hm	1. okt 2007		rev 1.1
	added compatibility to STEP7

*)
END_FUNCTION

(* POU leap_of_Date, ST *)
FUNCTION leap_of_Date : BOOL
VAR_INPUT
	idate : DATE;
END_VAR
VAR
END_VAR

(*
version 1.1	2 oct 2006
programmer 	hugo
tested by		tobias


leap_year is true if the tested year is a leap year  
execution time on wago 750-841 =  30 us   
*)
leap_of_Date := leap_year(year(idate));


(* change history

2.10.2006		changes to rev 1.1
the function now calls leap_year to accomodate further accuracy.
the function now works for any year from 1970 to 2100

*)
END_FUNCTION

(* POU leap_year, ST *)
FUNCTION leap_year : BOOL
VAR_INPUT
	yr : INT;
END_VAR
VAR
END_VAR

(*
version 1.1	2 oct 2006
programmer 	hugo
tested by		tobias


leap_year is true if the tested year is a leap year  
execution time on wago 750-841 =  12 us    
*)
leap_year := SHL(yr,14) = 0;

(* this code was used prior to rev 1.1

IF yr MOD 400 = 0 THEN leap_year := TRUE;
ELSIF yr MOD 100 = 0 THEN leap_year := FALSE;
ELSIF yr MOD 4 =0 THEN leap_year := TRUE;
ELSE leap_year := FALSE;
END_IF;

*)

(* change history

hm 	2.10.2006		rev 1.1
	the function now works for any year from 1970 up to 2100

hm	1. oct 2007		rev 1.2
	chaged code for higher performance
*)
END_FUNCTION

(* POU set_Date, ST *)
FUNCTION set_Date : DATE
VAR_INPUT
	year : INT;
	month : INT;
	day : INT;
END_VAR
VAR
	count : DWORD;
	leap: BOOL;
END_VAR

(*
version 1.2	1 okt 2007
programmer 	hugo
tested by		tobias

creates a date output from year, month and day of month   

*)
leap := leap_year(year);
IF STEP7 THEN
	count := TRUNC((year-1)*365.25-726483+day);
ELSE
	count := TRUNC((year-1)*365.25-719178+day);
END_IF;
CASE month OF
2:	count := count + 31;
3:	IF leap THEN count := count + 60; ELSE count := count + 59; END_IF;
4:	IF leap THEN count := count + 91; ELSE count := count + 90; END_IF;
5:	IF leap THEN count := count + 121; ELSE count := count + 120; END_IF;
6:	IF leap THEN count := count + 152; ELSE count := count + 151; END_IF;
7:	IF leap THEN count := count + 182; ELSE count := count + 181; END_IF;
8:	IF leap THEN count := count + 213; ELSE count := count + 212; END_IF;
9:	IF leap THEN count := count + 244; ELSE count := count + 243; END_IF;
10:	IF leap THEN count := count + 274; ELSE count := count + 273; END_IF;
11:	IF leap THEN count := count + 305; ELSE count := count + 304; END_IF;
12:	IF leap THEN count := count + 335; ELSE count := count + 334; END_IF;
END_CASE;
set_Date := DWORD_TO_DATE(count * 86400);


(* revision history
hm	4. aug. 2006	rev 1.0
	original version

hm	19 sep. 2007	rev 1.1
	use function leap_year to calculate leap year, more exceptions are handled

hm	1. okt	2007	rev 1.2
	added compatibilkity to step7
*)
END_FUNCTION

(* POU day_of_month, ST *)
FUNCTION day_of_month : INT
VAR_INPUT
	idate : DATE;
END_VAR
VAR
	yd: INT;
END_VAR

(*
version 1.3	8. okt 2007
programmer 	hugo
tested by		tobias

returns the day OF month for any DATE

*)
yd := day_of_year(idate);
IF leap_of_Date(idate) THEN
	CASE yd OF
		1..31 	:	day_of_month := yd;
		32..60	:	day_of_month := yd - 31;
		61..91	:	day_of_month := yd - 60;
		92..121 :	day_of_month := yd - 91;
		122..152:	day_of_month := yd - 121;
		153..182:	day_of_month := yd - 152;
		183..213:	day_of_month := yd - 182;
		214..244:	day_of_month := yd - 213;
		245..274:	day_of_month := yd - 244;
		275..305:	day_of_month := yd - 274;
		306..335:	day_of_month := yd - 305;
		336..366:	day_of_month := yd - 335;
	END_CASE;
ELSE
	CASE yd OF
		1..31 	:	day_of_month := yd;
		32..59	:	day_of_month := yd - 31;
		60..90	:	day_of_month := yd - 59;
		91..120 :	day_of_month := yd - 90;
		121..151:	day_of_month := yd - 120;
		152..181:	day_of_month := yd - 151;
		182..212:	day_of_month := yd - 181;
		213..243:	day_of_month := yd - 212;
		244..273:	day_of_month := yd - 243;
		274..304:	day_of_month := yd - 273;
		305..334:	day_of_month := yd - 304;
		335..365:	day_of_month := yd - 334;
	END_CASE;
END_IF;


(*
this function is simple but took too long with 133 us
the problem is date_to_string is far too slow
day_of_month := STRING_TO_INT(RIGHT(DATE_TO_STRING(idate),2));

Revision history

hm 22.1.2007		rev 1.1
	deleted unused variable day_in_year and day_in_year_begin

hm	1. okt 2007		rev 1.2
	changed code to use day_of_year and leap_of_date
	added compatibility to STEP7

hm	8. oct 2007		rev 1.3
	deleted unused variable yr
*)
END_FUNCTION

(* POU days_delta, ST *)
FUNCTION days_delta : INT
VAR_INPUT
	date_1 : DATE;
	date_2 : DATE;
END_VAR
VAR
END_VAR

(*
version 1.1	27 dec 2006
programmer 	hugo
tested by		tobias

days_delta calculates the days between two dates. the days are calculated date_2 - date_1.

*)
days_delta := day_of_date(date_2) - day_of_date(date_1);

(* revision history
hm	27. dec 2006	rev 1.0
	original version

hm	16.9.2007		rev 1.1
	coorected an error in formula and changed algorithm to show positive and negative delta

*)
END_FUNCTION

(* POU day_of_date, ST *)
FUNCTION day_of_date : INT
VAR_INPUT
	idate : DATE;
END_VAR
VAR
END_VAR


(*
	version 1.0	16 sep 2007
	programmer 	oscat
	tested BY		oscat

DAY_OF_DATE returns the days since 1.1.1970

*)
IF STEP7 THEN
	(* adjust step7 day by 7305 days because step7 date fornat starts at 1.1.1990  *)
	day_of_date := DWORD_TO_INT(DATE_TO_DWORD(idate) / 86400) + 7305;
ELSE
	day_of_date := DWORD_TO_INT(DATE_TO_DWORD(idate) / 86400);
END_IF;
(* revision history
hm		16.9.2007		rev 1.0
	original version

hm		1. okt 2007		rev 1.1
	added step7 compatibility

*)
END_FUNCTION

(* POU DST, ST *)
FUNCTION DST : BOOL
VAR_INPUT
	utc : DT;
	time_zone_offset : TIME;
END_VAR
VAR
	yr : INT;
	yr4 : DWORD;
	ltc: DWORD;
	idate : DWORD;
END_VAR

(*
version 1.0	4 aug 2006
programmer 	hugo
tested by		tobias

 this functions returns TRUE IF dst TIME is active 
 the FUNCTION calculates automaticall FOR any year betweek 1970 AND 2099 
wheather daylight savings is on OR off 
the summertime calculation is done according to european standards.
dst will become TRUE AT 02:00 in the morning FOR the respective days 
AND it will become FALSE after daylight savings TIME is switched back end OF october automatically 
(execution TIME on wago 750-841 =  110us   
*)
yr := year(DT_TO_DATE(utc));
ltc := DT_TO_DWORD(utc+time_zone_offset);
idate := DT_TO_DWORD(set_DT(yr,3,31,2,0,0));
yr4 := 5*yr/4;
IF idate - ((yr4+4) MOD 7)*86400 <= ltc AND idate + (214 - (yr4+1) MOD 7)*86400 > ltc THEN DST := TRUE; ELSE DST := FALSE; END_IF;


(*

Equation used TO calculate the beginning OF European Summer TIME:
Sunday (31 - (5*y/4 + 4) mod 7) March at 01.00 UTC
(valid through 2099, courtesy of Robert H. van Gent, EC).

European Summer Time ends (clocks go back) at 01.00 UTC on

    * 29 October 2006
    * 28 October 2007
    * 26 October 2008

Equation used to calculate the end of European Summer Time:
Sunday (31 - (5*y/4 + 1) mod 7) October at 01.00 UTC
(validity AND credits as above).

*)
END_FUNCTION

(* POU set_DT, ST *)
FUNCTION set_DT : DT
VAR_INPUT
	year : INT;
	month : INT;
	day : INT;
	hour : INT;
	minute : INT;
	second : INT;
END_VAR
VAR
END_VAR

(*
version 1.3	8 okt 2007
programmer 	hugo
tested by		tobias


creates a date output from year, month and day of month
year must be in the form of 4 digits ie 2006 or 1977.
execution time on wago 750-841 = 45 us   
*)
set_DT := DWORD_TO_DT(DATE_TO_DWORD(set_Date(year, month, day)) + second + minute * 60 + hour * 3600);


(* revision history
hm	4. aug. 2006	rev 1.0
	original version

hm	19 sep. 2007	rev 1.1
	use function leap_year to calculate leap year, more exceptions are handled

hm	1. okt 2007		rev 1.2
	added step7 compatibility
	call function set_date

hm	8. oct 2007		rev 1.3
	deleted unused variables count and leap
*)
END_FUNCTION

(* POU hour, ST *)
FUNCTION hour : INT
VAR_INPUT
	itod : TOD;
END_VAR
VAR
END_VAR

(*
version 1.1	2 okt 2006
programmer 	hugo
tested by		tobias

extracts the hour of a Time_of_day 
*)
hour := DWORD_TO_INT(TOD_TO_DWORD(itod)/3600000);


(* change history
hm 4. aug 2006	rev 1.0
	original version

hm 2.10.2006 	rev 1.1
	changed name of input to itod

*)
END_FUNCTION

(* POU minute, ST *)
FUNCTION minute : INT
VAR_INPUT
	itod : TOD;
END_VAR
VAR
END_VAR

(*
version 1.1	2 oct 2006
programmer 	hugo
tested by		tobias

extracts the minutes out of TOD truncating the ceconds 
execution time on wago 750-841  = 18us

*)  
minute := DWORD_TO_INT(TOD_TO_DWORD(itod)/60000 - TOD_TO_DWORD(itod)/3600000 * 60);


(* change history

2.10.2006 changes name of input to itod

*)
END_FUNCTION

(* POU second, ST *)
FUNCTION second : REAL
VAR_INPUT
	itod : TOD;
END_VAR
VAR
END_VAR

(*
version 1.1	2 oct 2006
programmer 	hugo
tested by		tobias

returns the seconds and milliseconds as real of TOD   
execution time on wago 750-841 = 20 us 
*)
second := DWORD_TO_REAL(TOD_TO_DWORD(itod) - TOD_TO_DWORD(itod)/60000 * 60000)/1000;



(* change history

2.10.2006 changes name of input to itod

*)
END_FUNCTION

(* POU easter, ST *)
FUNCTION easter : DATE
VAR_INPUT
	year : INT;
END_VAR
VAR
	A: INT;
	B: INT;
	C: INT;
	D: INT;
	e: INT;
	f: INT;
	g: INT;
	h: INT;
	i: INT;
	k: INT;
	l: INT;
	m: INT;
	n: INT;
	o: INT;
END_VAR

(*
version 1.0	27 dec 2006
programmer 	hugo
tested by		tobias

easter calculates the day of easter sunday for a given year.
most other catholic holidays are calculated in reference to easter sunday.

*)
a := year MOD 19;
b := year / 100;
c := year MOD 100;
d := b / 4;
e := b MOD 4;
f :=	(b + 8) / 25;
g := (b - f + 1) / 3;
h := (19 * a + b - d - g + 15) MOD 30;
i :=	c / 4;
k := c MOD 4;
l := (32 + 2 * e + 2 * i - h - k) MOD 7;
m := (a + 11 * h + 22 * l) / 451;
n := (h + l - 7 * m + 114) / 31;
o := (h + l - 7 * m + 114) MOD 31;

easter := set_Date(year,n,o+1);

(*
Im Magazin "Nature" vom 20. April 1876 veröffentlichte ein anonymer Autor eine Tabelle mit Regeln zur Berechnung des (Gregorianischen) Ostersonntages des Jahres J. In Formeln ausgedrückt erhält man das Folgende:
a	=	J mod 19
b	=	int(J / 100)
c	=	J mod 100
d	=	int(b / 4)
e	=	b mod 4
f	=	int((b + 8) / 25)
g	=	int((b - f + 1) / 3
h	=	(19 · a + b - d - g + 15) mod 30
i	=	int(c / 4)
k	=	c mod 4
l	=	(32 + 2 · e + 2 · i - h - k) mod 7
m	=	int((a + 11 · h + 22 · l) / 451)
n	=	int((h + l - 7 · m + 114) / 31)
o	=	(h + l - 7 · m + 114) mod 31

n ist hierbei die Nummer des Monats, o + 1 die Nummer des Tages auf welchen der Ostersonntag im Jahr J fällt. Dieser Algorithmus kommt ohne Hilfszahlen aus.

*)
END_FUNCTION

(* POU hour_to_time, ST *)
FUNCTION hour_to_time : TIME
VAR_INPUT
	input : REAL;
END_VAR
VAR
END_VAR

(*
version 1.0	4 aug 2006
programmer 	hugo
tested by		tobias

converts an amount of hours in real to time
execution TIME on wago 750-841 =  17us
*)
hour_to_time := DWORD_TO_TIME(REAL_TO_DWORD(input * 3600000));
END_FUNCTION

(* POU hour_to_tod, ST *)
FUNCTION hour_to_tod : TOD
VAR_INPUT
	input : REAL;
END_VAR
VAR
END_VAR

(*
version 1.0	4 aug 2006
programmer 	hugo
tested by		tobias

converts an amount of hours in real to time of day 
execution time on wago 750-841 =  17us 
*)
hour_to_tod := DWORD_TO_TOD(REAL_TO_DWORD(input * 3600000));
END_FUNCTION

(* POU local_time, ST *)
FUNCTION local_time : DT
VAR_INPUT
	utc : DT;
	time_zone_offset : TIME;
	dst_enable: BOOL;
END_VAR
VAR
END_VAR

(*
version 1.1	2 oct 2006
programmer 	hugo
tested by		tobias

localtime calculates the local time according to DSTenable and time_zone_offset.
the dst input only tells the function the dst (daylight savings time) is enabled but the calculation for summertime on and off is done by the function itself.
this means the dst input only tells the function to switch summertime on and off automatically or not.
the function will switch to summertime automatically at the specified time end of march and back end of october.
the summertime calculation is done according to european standards.
the input is world time (UTC) and a given time_zone_offset for any time_zone.

execution time on wago 750-841 = 140 us   
*)
IF DST(utc,time_zone_offset) AND dst_enable THEN
	local_time := utc + time_zone_offset + T#1h;
ELSE
	local_time := utc + time_zone_offset;
END_IF;


(*

change history

2.10.2006 hm	rev 1.1
	corrected an error in the dst check for correct function

*)
END_FUNCTION

(* POU Ltime_to_UTC, ST *)
FUNCTION Ltime_to_UTC : DT
VAR_INPUT
	Ltime : DT;
	DST : BOOL;
	Time_Zone_Offset : TIME;
END_VAR
VAR
END_VAR

(*
version 1.0	5 jul 2007
programmer 	hugo
tested by		tobias

LTIME_TO_UTC calculates UTC (World Time) from a local time LTIME. utc is calculated by subtracting Time_Zone_Offset from ltime and if dst it true subtracting an additional hour from ltime.

*)
IF DST THEN Ltime_to_UTC := Ltime - Time_Zone_Offset - t#1h; ELSE Ltime_to_UTC := Ltime - Time_Zone_Offset; END_IF;



(* revision history
5.7.2007	rev 1.0		original version

*)
END_FUNCTION

(* POU Ltime, ST *)
FUNCTION_BLOCK Ltime
VAR_INPUT
	UTC : DT;
	dst_enable : BOOL;
	time_zone_offset : TIME;
END_VAR
VAR_OUTPUT
	local_DT : DT;
	DST_on : BOOL;
	wday : INT;
END_VAR
VAR
	time_adder : TIME := t#0s;
	next_check : DT := dt#1970-01-01-00:00:00;
	init: BOOL;
END_VAR

(*

version 1.3	18 Mar 2007
programmer 	oscat
tested by		tobias

ltime is a real time clock that uses the system rtc as utc time and calculates and given time zone.
the utc time is supplied on the input UTC.
according to the input variable time_zone_offset when the input dst_enable is true,
the dst on and off times are calculated by a formula for any given year and the time is advanced and reset by one hour
at 02:00 and 03:00 for the last sunday of march and last sunday of october.
the code is high performance and the rtc counts every second.
if more then one time zone is needed by the systen the clock can be started many times by placing more then one function block.

execution time on wago 750-841 = 20 us 
 
*)
IF utc > next_check THEN
	IF NOT init THEN
		local_dt := utc + time_zone_offset;
		init := TRUE;
	END_IF;
	next_check := DWORD_TO_DT(DT_TO_DWORD(utc) / 3600 * 3600 +3600);
	DST_on := DST(local_dt, time_zone_offset);
	IF DST_on AND dst_enable THEN time_adder := time_zone_offset + T#1h; ELSE time_adder := time_zone_offset; END_IF;
END_IF;
local_dt :=utc + time_adder;
wday := weekday(DT_TO_DATE(local_dt));

(* revision history

hm 2.10.2006	rev 1.1
	corrected an error where dst would be delayed by 0.1second

hm 17.1.2007	rev 1.2
	added utc input instead of internal sysrtcgettime because this would only work on wago.
	dst_enable would not be checked before dst would be enabled.

hm 18.3.2007	rev 1.3
	changed code, dst would not work during first cycle.

*)
END_FUNCTION_BLOCK

(* POU weekday, ST *)
FUNCTION weekday : INT
VAR_INPUT
	idate : DATE;
END_VAR
VAR
END_VAR

(*
version 1.1	21 aug 2006
programmer 	hugo
tested by		tobias

calculates the weekday of a week   
monday = 1 ..... sunday = 7  

*)
weekday := DWORD_TO_INT((DATE_TO_DWORD(idate)/86400+3) MOD 7)+1;

(* revision history
hm 21.8.06 rev 1.1
	corrected a miscalculation formula is now correct 

*)
END_FUNCTION

(* POU minute_to_time, ST *)
FUNCTION minute_to_time : TIME
VAR_INPUT
	input : REAL;
END_VAR
VAR
END_VAR

(*
version 1.0	4 aug 2006
programmer 	hugo
tested by		tobias

converts an amount of minutes in real to time
execution time on wago 750-841 =  17us
*) 
minute_to_time := DWORD_TO_TIME(REAL_TO_DWORD(input * 60000));
END_FUNCTION

(* POU multime, ST *)
FUNCTION multime : TIME
VAR_INPUT
	t : TIME;
	M : REAL;
END_VAR
VAR
END_VAR


(*
version 1.0	2 oct 2006
programmer 	hugo
tested by		tobias

multiplies a time by a real number and returns a time
*)
multime := REAL_TO_TIME(TIME_TO_REAL(t)*M);
END_FUNCTION

(* POU second_to_time, ST *)
FUNCTION second_to_time : TIME
VAR_INPUT
	input : REAL;
END_VAR
VAR
END_VAR

(*
version 1.0	4 aug 2006
programmer 	hugo
tested by		tobias

converts an amount of seconds in real to time
execution TIME on wago 750-841 =  17us 

*)
second_to_time := DWORD_TO_TIME(REAL_TO_DWORD(input * 1000));
END_FUNCTION

(* POU set_Tod, ST *)
FUNCTION set_Tod : TOD
VAR_INPUT
	hour : INT;
	minute : INT;
	second : REAL;
END_VAR
VAR
END_VAR

(*
version 1.0	4 aug 2006
programmer 	hugo
tested by		tobias

creates tod from hour minute and second 
execution time on wago 750-841 = 14 us  
*)
set_Tod := DWORD_TO_TOD(DINT_TO_DWORD(TRUNC(second * 1000) + minute * 60000 + hour * 3600000));

(* revision history

hm	4.aug.2006
	original version

hm	11. sep 2007
	changed coding to avoid a compiler warning under twincat.

*)
END_FUNCTION

(* POU work_week, ST *)
FUNCTION work_week : INT
VAR_INPUT
	idate : DATE;
END_VAR
VAR
	wday1 : INT;
END_VAR

(*
version 1.1	14 jan 2007
programmer 	hugo
tested by		tobias

calculates the work week for a given date  
execution time on wago 750-841 = 155us   
*)
wday1 := weekday(set_Date(year(idate), 1,1));
IF wday1 < 5 THEN
	work_week := TRUNC((day_of_year(idate) + wday1 + 5)/7);
ELSE
	work_week := TRUNC((day_of_year(idate) + wday1 - 2)/7);
END_IF


(* revision history

hm 17.1.2007		rev 1.1
	deleted unused variable yday

*)
END_FUNCTION

(* POU T_PLC_US, ST *)
FUNCTION T_PLC_US : DWORD
VAR CONSTANT
	debug : BOOL := FALSE;
	N : INT := 0;
	offset : DWORD := 0;
END_VAR
VAR
	temp : DWORD := 1;
END_VAR

(*
version 1.0	14 sep 2007
programmer 	hugo
tested by		tobias

T_PLC_US reads the internal PLC timer and return the time, it has the advantage to be able to set a debug mode 
and speed up the counter to test the plc timer overrun which occurs every 50 days respectively 25 days at siemens S7
this routine also allows to correct the behavior of s7 where the internal plc counter will not count all 32 bits.

*)
T_PLC_US := TIME_TO_DWORD(TIME())*1000;
(* hier muss die korrektur für step7 stattfinden
plctime muss den vollen wertebereich von time ausnutzen:
wenn bei step7 time -24tage bis plus 24 tage ist dann muss der timer auch beim überlauf auf -24tage springen 
und auf keinen fall auf 0 !!!!
für siemens muss ein weiterer fb im main eingebunden werden der sicherstellt das alle 32 bits durchgezählt werden.
es kann nur ein fb sein den er muss sich das oberste (32te) bit merken.
oder etwa spring s7 bei überlauf auf -24 tage????? dann wäre keine korrektur nötig.
*)
IF debug THEN
	T_PLC_US := (SHL(T_PLC_US,N) OR SHL(temp,N)-1) + Offset;
END_IF;

(* revision history
hm	14.9.2007	rev 1.0
	original version

*)
END_FUNCTION

(* POU SHR1, ST *)
FUNCTION SHR1 : DWORD
VAR_INPUT
	IN : DWORD;
	N : INT;
END_VAR
VAR CONSTANT
	temp : DWORD := 2#11111111_11111111_11111111_11111111;
END_VAR

(*
version 1.0	14 sep 2007
programmer 	hugo
tested by		tobias

SHR1 shifts N bits to the right filling the new bits with 1

*)
IF N = 0 THEN
	SHR1 := in;
ELSE
	SHR1 := SHR(IN,N) OR SHL(temp,32-N);
END_IF;

(* revision history
hm	14.9.2007	rev 1.0
	original version

*)
END_FUNCTION

(* POU SHL1, ST *)
FUNCTION SHL1 : DWORD
VAR_INPUT
	IN : DWORD;
	N : INT;
END_VAR
VAR CONSTANT
	temp : DWORD := 1;
END_VAR

(*
version 1.0	14 sep 2007
programmer 	hugo
tested by		tobias

SHL1 shifts N bits to the left filling the new bits with 1

*)
IF N = 32 THEN
	SHL1 := 16#FF_FF_FF_FF;
ELSE
	SHL1 := SHL(IN,N) OR SHL(temp,N)-1;
END_IF;

(* revision history
hm	14.9.2007	rev 1.0
	original version

*)
END_FUNCTION

(* POU period, ST *)
FUNCTION period : BOOL
VAR_INPUT
	d1 : DATE;
	dx : DATE;
	d2 : DATE;
END_VAR
VAR
	p1 : DATE;
	p2 : DATE;
	yx: INT;
END_VAR

(*
version 1.1	20 sep 2007
programmer 	hugo
tested by		tobias

PERIOD checks if a given date is between two dates (d1 and d2) d1 is the starting date and d2 the last date for the period.
the years of the dates are ignored, so the function period cheks for a time period within a year independet of the year.

*)
yx := year(dx);
p1 := date_add(d1,0,0,0,yx - year(d1));
p2 := date_add(d2,0,0,0,yx - year(d2));

IF p2 >= p1 THEN
	period := dx <= p2  AND dx >= p1;
ELSE
	period := dx <= p2 OR dx >= p1;
END_IF;

(* revision history

hm		19. sep 2007		rev 1.0
	original version

hm		20. sep 2007		rev 1.1
	corrected a problem with leap year

*)
END_FUNCTION

(* POU HEX_TO_DWORD, ST *)
FUNCTION HEX_TO_DWORD : INT
VAR_INPUT
	Hex : STRING;
END_VAR
VAR
	pt : POINTER TO BYTE;
	i: INT;
	X: BYTE;
END_VAR

(*
version 1.0	6 oct 2006
programmer 	hugo
tested by		tobias

HEX_TO_DWORD converts a Hexadecimal string into a DWORD.

*)
pt := ADR(hex);
FOR I := 1 TO LEN(hex) DO
	x := pt^ - 48;
	IF X > 9 THEN X := X - 7; END_IF;
	HEX_TO_DWORD := SHL(HEX_TO_DWORD,4) + X;
	pt := pt + 1;
END_FOR

(* revision histroy
hm		2.10.2007		rev 1.0
	original release

*)	
END_FUNCTION

(* POU FT_rmp, ST *)
FUNCTION_BLOCK FT_rmp
VAR_INPUT
	Rmp : BOOL := TRUE;
	in : REAL;
	KR : REAL;
	KF : REAL;
END_VAR
VAR_OUTPUT
	out : REAL;
	busy : BOOL;
	UD : BOOL;
END_VAR
VAR
	tx: TIME;
	last: TIME;
	init: BOOL;
END_VAR

(*
	version 1.3	17 sep 2007
	programmer 	oscat
	tested BY		oscat

this ramp function follows an input signal with a linear ramp up or down, the up or down speed can be set with KF and KR.
a K factor of 1 means 1 unit per second on the output. K factors can only be positive and not negative.
a busy output signals the ramp is running or busy false means the in value is present on the output.
a rmp input false means the output follows the input dierctly while a rmp = true means the output follows the input with a ramp.
a updn output signal the directon of the ramp (up or down).

*)
(* read system time *)
tx := DWORD_TO_TIME(T_PLC_MS()) - last;

IF NOT init THEN
	init := TRUE;
	last := tx;
	tx := t#0s;
	out := in;
END_IF;
IF NOT rmp THEN
	out := in;
	busy := FALSE;
ELSIF out > in AND kf > 0 THEN
	(* ramp down *)
	out := out - TIME_TO_REAL(tx) / 1000 * KF;
	IF out < in THEN out := in; END_IF;
ELSIF out < in AND kr > 0 THEN
	(* ramp up *)
	out := out + TIME_TO_REAL(tx) / 1000 * KR;
	IF out > in THEN out := in; END_IF;
END_IF;

(* set busy and dir flags *)
IF out < in THEN
	busy := TRUE;
	ud := 1;
ELSIF out > in THEN
	busy := TRUE;
	ud := 0;
ELSE
	busy := FALSE;
END_IF;
last := last + tx;


(* revision history:

hm 8.10.2006			rev 1.1
	added ud output

hm 12. feb 2007		rev 1.2
	added init variable and corrected a possible startup problem

hm	17. sep 2007	rev 1.3
	replaced time() with t_plc_ms() for compatibility reasons

*)
END_FUNCTION_BLOCK

(* POU SPLINE_INT, ST *)
FUNCTION_BLOCK SPLINE_INT
VAR_INPUT
	X : REAL;
END_VAR
VAR_OUTPUT
	Y : REAL;
END_VAR
VAR CONSTANT
	n : INT := 5;
END_VAR
VAR
	Xs : ARRAY[1..n] OF REAL;
	Ys : ARRAY[1..n] OF REAL;
	I, J : INT;
	init: BOOL;
END_VAR
RETURN;
END_FUNCTION_BLOCK

(* POU Pulse_Length, ST *)
FUNCTION_BLOCK Pulse_Length
VAR_INPUT
	in : BOOL;
END_VAR
VAR_OUTPUT
	short : BOOL;
	middle : BOOL;
	long : BOOL;
END_VAR
VAR_INPUT CONSTANT
	T_short : TIME := t#100ms;
	T_long : TIME := t#1s;
END_VAR
VAR
	tx : TIME;
	tn: TIME;
	edge : BOOL;
END_VAR

(*
version 1.1	15 sep 2007
programmer 	oscat
tested by		tobias

Pulse_length indicates on 3 outputs if an input pulse had been shorter than T_short (short = True), longer than T_long (long = True) or between T_short and T_long (middle = True).

*)
(* read system time *)
tx := DWORD_TO_TIME(T_PLC_MS());

(* reset outputs, they should only be active 1 cycle *)
short := FALSE;
Middle := FALSE;
long := FALSE;

(* detect rising edge *)
IF in AND NOT edge THEN
	edge := TRUE;
	tn := tx;

(* detect for falling edge *)
ELSIF NOT in AND edge THEN
	edge := FALSE;
	tn := tx - tn;
	IF tn < t_short THEN
		short := TRUE;
	ELSIF tn > t_long THEN
		long := TRUE;
	ELSE
		Middle := TRUE;
	END_IF;

(* generate long pulse as soon as T_long is reached *)
ELSIF in AND tx - tn > t_long THEN
	long := TRUE;
END_IF;


(* revision history

hm	15. feb 2006	rev 1.0
	original version

hm	15 sep 2007		rev 1.1
	replaced Time() with T_PLC_MS for compatibility and performance reasons

*)
END_FUNCTION_BLOCK

(* POU TOGGLE, ST *)
FUNCTION_BLOCK TOGGLE
VAR_INPUT
	CLK : BOOL;
	rst : BOOL := FALSE;
END_VAR
VAR_OUTPUT
	Q : BOOL;
END_VAR
VAR
	edge : BOOL;
END_VAR

(*
version 1.0	13 sep 2007
programmer 	hugo
tested by		tobias

toggle flip flop the output changes state with every rising edge of clk.

*)
IF rst THEN
	q := 0;
ELSIF clk AND NOT edge THEN
	Q := NOT Q;
END_IF;
edge := clk;

(* revision history

hm	13.9.2007		rev 1.0
	original version

*)
END_FUNCTION_BLOCK

(* POU LINEAR_INT, ST *)
FUNCTION LINEAR_INT : REAL
VAR_INPUT
	X : REAL;
	XY : ARRAY[1..20,0..1] OF REAL;
	Pts : INT;
END_VAR
VAR
	i : INT;
END_VAR

(*
	version 1.0	7 oct 2007
	programmer 	oscat
	tested BY		oscat

LINEAR_INT calculates an output based on a linear interpolation of up to 20 coordinates given in an array
the indut coordinates have to start at the lowest array position and must be sorted ba ascending X values.

*)
(*make sure n is bound within the array size *)
IF pts > 20 THEN pts := 20; END_IF;

(* calculate the linear segement interpolation *)
I := 2;
(* search for segment and calculate output
	below and above the defined segments we interpolate the last segment *)
WHILE (i < pts) AND (XY[i,0] < X) DO
	i := i + 1;
END_WHILE;

(* calculate the output value on the corresponding segment coordinates *)
LINEAR_INT := ((XY[i,1] - XY[i-1,1]) * X - XY[i,1] * XY[i-1,0] + XY[i-1,1]*XY[i,0]) / (XY[i,0] - XY[i-1,0]);

(* revision history
hm	7. oct 2007		rev 1.0
	original version

*)
END_FUNCTION

(* POU POLYNOM_INT, ST *)
FUNCTION POLYNOM_INT : REAL
VAR_INPUT
	X : REAL;
	XY : ARRAY[1..5,0..1] OF REAL;
	Pts : INT;
END_VAR
VAR
	I, J : INT;
	init: BOOL;
END_VAR

(*
	version 1.0	7 oct 2007
	programmer 	oscat
	tested BY		oscat

POLYNOM_INT calculates an output based on a Polynom interpolation of up to 5 coordinates given in an array
the indut coordinates have to start at the lowest array position and must be sorted ba ascending X values.

*)
(*make sure n is bound within the array size *)
IF pts > 5 THEN pts := 5; END_IF;

(* this part is only to calculate the polynom parameters, which are then stores in the Y array
	the array values, it is not needed during runtime, unless the parameters will change during runtime
	the remaining code without this setup code can be used within a function to calculate specific functions
	the content of the arrays is then used as constant values within the function *)
IF NOT init THEN
	init := TRUE;
	FOR i := 1 TO pts DO
       	FOR j := pts TO i + 1 BY -1 DO
           		XY[j,1] := (XY[j,1] - XY[j-1,1]) / (XY[j,0] - XY[j-i,0]);
		END_FOR;
	END_FOR;
END_IF;

(* this part is the actual calculation *)
POLYNOM_INT := 0;
FOR i := pts TO 1 BY -1DO
       POLYNOM_INT := POLYNOM_INT * (X - XY[i,0]) + XY[i,1];
END_FOR;


(* revision history
hm		8. okt 2007	rev 1.0
	original version

*)
END_FUNCTION

(* POU crc_test, CFC *)
PROGRAM crc_test
VAR
	arr : ARRAY[1..9] OF BYTE := 49, 50, 51, 52, 53, 54, 55, 56, 57;
	code: DWORD;
	hex: STRING;
END_VAR
VAR (* helpers for the ST form of the networks *)
	_t1 : DWORD;
END_VAR
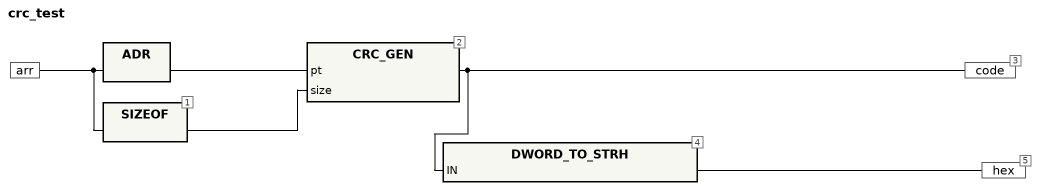
_CFC_ (* Continuous Function Chart, elements in execution order *)
#0 ADR(arr)
#1 SIZEOF(arr)
#2 CRC_GEN(pt: #0, size: #1, Polynom_L := 263, init := 255, XOR_out := 255, rev_in := TRUE, rev_out := TRUE)
#3 code <= #2
#4 DWORD_TO_STRH(IN: #2)
#5 hex <= #4
_END_CFC_
(* the same logic as Structured Text *)
_t1 := CRC_GEN(ADR(arr), SIZEOF(arr));
code := _t1;
hex := DWORD_TO_STRH(IN := _t1);
END_PROGRAM

(* POU blind_test, CFC *)
PROGRAM blind_test
VAR
	up: BOOL;
	dn: BOOL;
	x1: blind_actuator;
	mu: BOOL;
	md: BOOL;
	pos: BYTE;
	ang: BYTE;
	x2: blind_security;
	esr: BYTE;
	fire: BOOL;
	wind: BOOL;
	alarm: BOOL;
	rain: BOOL;
	x3: blind_control;
	p_set: BYTE;
	a_set: BYTE;
	sens: BYTE;
	x5: blind_input;
	auto: BOOL;
	p: BYTE;
	a: BYTE;
	Manual: BOOL;
	Input: BOOL;
	IN: BOOL;
	x6: sun_pos;
	lat: REAL;
	lon: REAL;
	utc: DT;
	sun: BOOL;
	X7: blind_night;
	x8: sun_time;
	Door: BOOL;
	pres: BOOL;
	td: TIME;
END_VAR
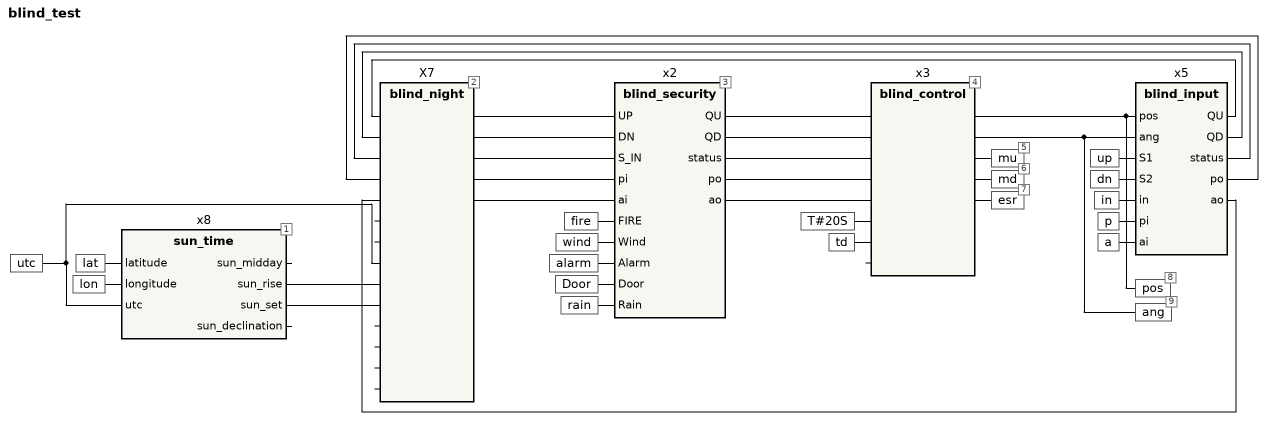
_CFC_ (* Continuous Function Chart, elements in execution order *)
#0 x5:blind_input(pos: #4.out 1, ang: #4.out 2, S1: up, S2: dn, in: in, pi: p, ai: a, click_mode := TRUE, click_time := T#250ms, manual_timeout := T#10s)
#1 x8:sun_time(latitude: lat, longitude: lon, utc: utc)
#2 X7:blind_night(#0.QU, #0.QD, #0.status, #0.po, #0.ao, -, -, utc, #1.sun_rise, #1.sun_set, -, -, -, -)
#3 x2:blind_security(UP: #2.out 1, DN: #2.out 2, S_IN: #2.out 3, pi: #2.out 4, ai: #2.out 5, FIRE: fire, Wind: wind, Alarm: alarm, Door: Door, Rain: rain)
#4 x3:blind_control(#3.QU, #3.QD, #3.status, #3.po, #3.ao, T#20S, td, -, sens := 5)
#5 mu <= #4.out 3
#6 md <= #4.out 4
#7 esr <= #4.out 5
#8 pos <= #4.out 1
#9 ang <= #4.out 2
_END_CFC_
END_PROGRAM

(* POU blind_actuator, ST *)
 FUNCTION_BLOCK blind_actuator
VAR_INPUT
	UP, DN : BOOL;
	S_IN : BYTE;
	T_UD : TIME := T#10s;
	T_Angle : TIME := T#3s;
END_VAR
VAR_INPUT CONSTANT
	T_lockout : TIME := t#100ms;
END_VAR
VAR_OUTPUT
	pos, ang : BYTE;
	QU, QD : BOOL;
	status : BYTE;
END_VAR
VAR
	position, angle : rmp_B;
	lock : interlock;
END_VAR

(*
version 1.1	6 oct 2007
programmer 	hugo
tested by		tobias

blind actuator drives the up and down motor of a blind. T_lockout specifies the time between up or dn becomes active. 
To change direction there must be a minimum wait time to allow the motors to come to rest first.
the up and down outputs QU and QD are controlled by the inputs UP and DN.
the outputs pos and ang simulate the position of the blind pos = 0 means blind is down and pos = 255 = blind is up.
the angle 0 means vertical posisition of the slates and 255 means horizontal position of the slates.


*)
(* make sure only one motor is active at a given time *)
lock(i1 := UP, I2 := DN, TL := T_lockout);

(* ramp up or down to simulate the angle position of the blind slats *)
angle(en := lock.Q1 OR lock.Q2, UP := lock.Q1, PT := T_Angle);
position(en := lock.Q1 AND angle.high OR lock.Q2 AND angle.low, up := lock.Q1, PT := T_UD);

(* set the outputs *)
pos := position.Out;
ang := angle.Out;
QU := lock.Q1;
QD := lock.Q2;

(* set the status output *)
IF UP AND DN THEN
	IF s_in < 10 AND S_in > 1 THEN status := s_in; ELSE status := 1; END_IF;			(* error up and down together are not allowed *)
ELSIF S_IN > 0 THEN
	status := S_IN;
ELSIF UP THEN
	status := 101;
ELSIF DN THEN
	status := 102;
ELSE
	status := 0;
END_IF;


(* revision history
hm	29. sep 2007	rev 1.0
	original release

hm	6. oct 2007		rev 1.1
	rearranged outputs
	
*)
END_FUNCTION_BLOCK

(* POU rmp_B, ST *)
FUNCTION_BLOCK rmp_B
VAR_INPUT
	SET : BOOL := FALSE;
	PT : TIME;
	EN : BOOL := TRUE;
	UP : BOOL := TRUE;
	RST : BOOL := FALSE;
END_VAR
VAR_OUTPUT
	out : BYTE;
	busy: BOOL;
	high : BOOL;
	low : BOOL;
END_VAR
VAR
	last_step : DWORD;
	now : DWORD;
	tmp: DWORD;
	edge: BOOL;
	N : BYTE;
END_VAR

(*
	version 1.5	5 oct 2007
	programmer 	oscat
	tested BY		oscat

this ramp generator generates a byte wide ramp with 255 steps
the generator has an asynchronous set and reset
the ramp is controlled by PT which is the total ramp time for a full sweep from 0..255
an UD input controlls the direction Up or Down and the E input enables the ramp generation
a busy output indicates that the ramp is running, busy false means output is stable.
the outputs low and high will be true when the output has reached its max or min value.

*)
(* read system time *)
now := T_PLC_US();

(* calculate the necessary step response *)
IF pt = t#0s THEN
	tmp := 255;
ELSE
	tmp := SHL(now - last_step, 8) / (TIME_TO_DWORD(pt)*1000);
END_IF;
IF tmp > 255 THEN N:= 255; ELSE N:= DWORD_TO_BYTE(tmp); END_IF;

(* detetct edge on en *)
IF en AND NOT edge THEN
	last_step := now;
(* check for asynchronous set or reset *)
ELSIF rst THEN
	out := 0;
ELSIF set  THEN
	out := 255;
ELSIF en AND N > 0 THEN
	(* generate ramp *)
	last_step := last_step + SHR(N * TIME_TO_DWORD(pt) * 1000,8);
	IF UP THEN
		IF out > 255 - N THEN out := 255; ELSE out := out + N; END_IF;
	ELSE
		IF out < N THEN out := 0; ELSE out := out - N; END_IF;
	END_IF;
END_IF;
edge := en;

(* checks for outputs stable and reset or set busy flag *)
IF out = 0 THEN
	busy := FALSE;
	low := TRUE;
	high := FALSE;
ELSIF out = 255 THEN
	busy := FALSE;
	high := TRUE;
	low := FALSE;
ELSE
	busy := en;
	high := FALSE;
	low := FALSE;
END_IF;


(* revision history

hm 5.10.2006	rev 1.1
	added busy output
hm 17.1.2007	rev 1.2
	renamed input ud to up for better usability
	deleted unused variable step

hm	17.9.2007	rev 1.3
	replaced time() with t_plc_ms() for compatibility reasons

hm	28. sep 2007	rev 1.4
	added outputs on and off
	busy is now disabled while en is false
	new coding for higher accuracy and performance

hm	5. oct 2007		rev 1.5
	added statements to allow for PT to be t#0s output jumps to max or min immediately

*)
END_FUNCTION_BLOCK

(* POU interlock, ST *)
FUNCTION_BLOCK interlock
VAR_INPUT
	I1, I2 : BOOL;
	TL : TIME;
END_VAR
VAR_OUTPUT
	Q1, Q2 : BOOL;
END_VAR
VAR
	T1, T2 : TOF;
END_VAR

(*
version 1.0	28 sep 2007
programmer 	hugo
tested by		tobias

INTERLOCK has two inputs I1 and I2 which drive the corresponding outputs Q1 and Q2.
the inputs signals lock each other out and therfore I1 can only drive Q1 when I2 is Low and vice versa.
The input TL specifies a dead time between two outputs can become active.
an output can only become active when the other output was not active for the time TL.

*)
(* the input signal have a run delay to lockout the other input *)
T1(IN := I1, PT := TL);
T2(IN := I2, PT := TL);

Q1 := I1 AND NOT t2.Q;
Q2 := I2 AND NOT t1.Q;


(* revision history

hm	28 sep 2007		rev 1.0
	original version

*)
END_FUNCTION_BLOCK

(* POU blind_security, ST *)
FUNCTION_BLOCK blind_security
VAR_INPUT
	UP, DN : BOOL;
	S_IN : BYTE;
	pi, ai : BYTE;
	FIRE : BOOL;
	Wind : BOOL;
	Alarm : BOOL;
	Door : BOOL;
	Rain : BOOL;
END_VAR
VAR_INPUT CONSTANT
	Alarm_UP : BOOL := TRUE;
END_VAR
VAR_OUTPUT
	QU, QD : BOOL;
	status : BYTE;
	po, ao : BYTE;
END_VAR
VAR
END_VAR

(*
version 1.1	6. oct 2007
programmer 	hugo
tested by		tobias


*)
IF Fire THEN
	QU := TRUE;
	QD := FALSE;
	status := 111;
ELSIF Wind THEN
	QU := TRUE;
	QD := FALSE;
	status := 112;
ELSIF alarm THEN
	QU := Alarm_up;
	QD := NOT Alarm_up;
	status := 113;
ELSIF Door THEN
	QU := TRUE;
	QD := FALSE;
	status := 114;
ELSIF Rain AND NOT (up XOR dn) THEN
	QU := FALSE;
	QD := TRUE;
	status := 115;
ELSE
	QU := UP;
	QD := DN;
	status := S_IN;
	po := pi;
	ao := ai;
END_IF;


(* revision history
hm	29. sep 2007	rev 1.0
	original release

hm	6. oct 2007		rev 1.1
	added pos and angle inputs and outputs
	manual will override rain position
	alarm position can now be configured

*)
END_FUNCTION_BLOCK

(* POU blind_control, ST *)
FUNCTION_BLOCK blind_control
VAR_INPUT
	UP, DN : BOOL;
	S_IN : BYTE;
	pi : BYTE;
	ai : BYTE;
	T_UD, T_ANGLE : TIME;
END_VAR
VAR_INPUT CONSTANT
	sens : BYTE;
END_VAR
VAR_OUTPUT
	pos, ang : BYTE;
	MU, MD : BOOL;
	status : BYTE;
END_VAR
VAR
	act : blind_actuator;
	delta : BYTE;
END_VAR

(*
version 1.1	6 oct 2007
programmer 	hugo
tested by		tobias


*)
IF UP AND DN THEN
	(* automatic modus detected *)
	(* first find regulate correct position *)
	IF BYTE_TO_INT(act.pos) < BYTE_TO_INT(pi) - delta THEN
		act.UP := TRUE;
		act.DN := FALSE;
		delta := 0;
		act.S_IN := 121;
	ELSIF BYTE_TO_INT(act.pos) > BYTE_TO_INT(pi) + delta THEN
		act.UP := FALSE;
		act.DN := TRUE;
		delta := 0;
		act.S_IN := 122;
	(* regulate angle *)
	ELSIF BYTE_TO_INT(act.ang) < BYTE_TO_INT(ai) - delta THEN
		act.UP := TRUE;
		act.DN := FALSE;
		delta := 0;
		act.S_IN := 123;
	ELSIF BYTE_TO_INT(act.ang) > BYTE_TO_INT(ai) + delta THEN
		act.UP := FALSE;
		act.DN := TRUE;
		delta := 0;
		act.S_IN := 124;
	(* correct position reached *)
	ELSE
		act.UP := FALSE;
		act.DN := FALSE;
		delta := sens;
		act.S_IN := 0;
	END_IF;
ELSE
	act.UP := UP;
	act.DN := DN;
END_IF;

(* hand over status *)
IF s_in > 0 THEN act.S_IN := S_IN; END_IF;

(* blind control calls blind_actuator *)
act(T_UD:=T_UD, T_ANGLE:=T_ANGLE);
pos := act.pos;
ang := act.ang;
MU := act.QU;
md := act.QD;
status := act.status;

(* revision history
hm	29. sep 2007	rev 1.0
	original release

hm	6. oct 2007		rev 1.1
	rearranged outputs
	integrated blind_actuator minto blind_control

*)
END_FUNCTION_BLOCK

(* POU blind_input, ST *)
FUNCTION_BLOCK blind_input
VAR_INPUT
	pos, ang : BYTE;
	S1, S2 : BOOL;
	in : BOOL;
	pi, ai : BYTE;
END_VAR
VAR_INPUT CONSTANT
	single_switch : BOOL := FALSE;
	click_mode : BOOL := TRUE;
	click_time : TIME := T#200ms;
	manual_timeout: TIME := T#1h;
END_VAR
VAR_OUTPUT
	QU, QD : BOOL;
	status : BYTE;
	po, ao : BYTE;
END_VAR
VAR
	tog1, tog2 : TOGGLE;
	pl1, pl2 : Pulse_Length;
	SU, SD : BOOL;
	last_act: DWORD;
	tx: DWORD;
END_VAR

(*
version 1.1	6 oct 2007
programmer 	hugo
tested by		tobias


*)
(* read system_time *)
tx := T_PLC_MS();

(* single or double switch operation *)
IF click_mode THEN
	PL1(in := S1, T_short := click_time, T_long := click_time);
	PL2(in := S2, T_short := click_time, T_long := click_time);
	tog1(clk := pl1.short, rst := pl1.long OR pl2.short OR pl2.long);
	tog2(clk := pl2.short, rst := pl2.long OR pl1.short OR pl1.long);
	SU := tog1.Q OR PL1.long;
	SD := tog2.Q OR pl2.long;
ELSE
	tog1(CLK := NOT S1);
	SU := (S1 AND NOT tog1.Q AND single_switch) OR (NOT single_switch AND S1);
	SD := (S1 AND tog1.Q AND single_switch) OR (NOT single_switch AND S2);
END_IF;

(* Forced Input is active *)
IF in THEN
	QU := TRUE;
	QD := TRUE;
	po := pi;
	ao := ai;
	status := 131;

(* in manual mode set ps and as to actual values *)
ELSIF SU OR SD THEN
	po := pos;
	ao := ang;
	last_act := tx;
	QU := SU;
	QD := SD;
	IF su THEN status := 132; ELSE status := 133; END_IF;

(* enable automatik mode after auto timer has expired *)
ELSIF manual_timeout > t#0s AND tx - last_act >= TIME_TO_DWORD(manual_timeout) THEN
	QU := TRUE;
	QD := TRUE;
	status := 134;

(* no input active *)
ELSE
	QU := FALSE;
	QD := FALSE;
	status := 0;
END_IF;


(* revision history
hm	29. sep 2007	rev 1.0
	original release

hm	6. oct 2007		rev 1.1
	renamed ps and as to po and ao

*)
END_FUNCTION_BLOCK

(* POU sun_pos, ST *)
FUNCTION_BLOCK sun_pos
VAR_INPUT
	latitude : REAL;				(* latitude of geographical position  *)
	longitude : REAL;				(* longitude of geographical position  *)
	utc : DT;						(*	world time				*)
END_VAR
VAR_OUTPUT
	B: REAL;
	HR: REAL;
END_VAR
VAR
	L: REAL;
	N: REAL; (* amount of days since 1.1.2000 12:00 *)
	G: REAL;
	K: REAL;
	A: REAL;
	X: REAL;
	D: REAL;
	JD: REAL;
	JD0: REAL;
	T: REAL;
	P: REAL;
	Ph: REAL;
	TA: REAL;
	H: REAL;
	RF: REAL;
	T1: REAL;
END_VAR

(*
version 1.0	1 Feb 2007
programmer 	hugo
tested by		tobias

this FUNCTION block calculates the sun position for a given date and time.
the times are calculated in utc and have to be corrected for the given time zone.
B is the angle from north and HR is the highth in degrees.

*)
N := (DT_TO_DWORD(utc) - 946728000)/86400.0;
JD := N + 2451545.0;
L := 280.460 + 0.9856474 * N;
L := modR(L,360);
G := 357.528 + 0.9856003 * N;
G := Rad(modR(G,360));
K := Rad(L + 1.915 * SIN(G) + 0.02 * SIN(2*G));
X := Rad(23.439 - 0.0000004 * N);
A := ATAN(COS(X)*SIN(K)/COS(K));
IF COS(K) < 0 THEN A := A + PI; END_IF;
D := ASIN(SIN(X) * SIN(K));
JD0 := TRUNC(JD - 0.5) + 0.5;
T := (TRUNC(N - 0.5) + 0.5) / 36525;
Ph := modR(6.697376 + 2400.05134 * T + 1.002738 * TOD_TO_REAL(DT_TO_TOD(utc))/3600000, 24);
P := PH * 15 + longitude;
TA := P - deg(A);
T1 := COS(Rad(TA))*SIN(Rad(latitude)) - TAN(D)*COS(Rad(latitude));
B := deg(ATAN(SIN(Rad(TA))/T1));
IF T1 < 0 THEN B := B + 180; END_IF;
IF B > 180 THEN
	B := B - 180;
ELSIF B < 180 THEN
	B := B + 180;
END_IF;
H := deg(ASIN(COS(D)*COS(Rad(TA))*COS(Rad(latitude))+SIN(D)*SIN(Rad(latitude))));
RF := 1.02 / TAN(Rad(H+10.3/(H+5.11)));
HR := H + RF / 60;
END_FUNCTION_BLOCK

(* POU blind_night, ST *)
FUNCTION_BLOCK blind_night
VAR_INPUT
	UP, DN : BOOL;
	S_IN : BYTE;
	pi, ai : BYTE;
	E_night : BOOL := TRUE;
	E_day	: BOOL := TRUE;
	dtin : DT;
	sunrise, sunset : TOD;
END_VAR
VAR_INPUT CONSTANT
	sunrise_offset : TIME;
	sunset_offset : TIME;
	night_position : BYTE := 0;
	night_angle : BYTE := 0;
END_VAR
VAR_OUTPUT
	QU, QD : BOOL;
	status : BYTE;
	po, ao : BYTE;
END_VAR
VAR
	night : BOOL;
	last_night, last_day : DATE;
END_VAR

(*
version 1.2	6 oct 2007
programmer 	hugo
tested by		tobias


*)
IF NOT (up AND dn) AND night THEN
	(* manual operation at night will cancel operation for one night *)
	night := FALSE;
ELSIF (DT_TO_TOD(dtin) > sunset + sunset_offset) AND (last_night < DT_TO_DATE(dtin)) AND NOT night AND e_night THEN
	(* enable night *)
	night := TRUE;
	last_night := DT_TO_DATE(dtin);
ELSIF (DT_TO_TOD(dtin) > sunrise + sunrise_offset) AND (last_day < DT_TO_DATE(dtin)) AND night AND e_day AND (last_night < DT_TO_DATE(dtin)) THEN
	(* disable night *)
	night := FALSE;
	last_day := DT_TO_DATE(dtin);
END_IF;

(* shade at night only in auto mode and enable = true *)
IF UP AND DN AND night THEN
	status := 141;
	po := night_position;
	ao := night_angle;
ELSE
	QU := UP;
	QD := DN;
	po := pi;
	ao := ai;
	status := s_in;
END_IF;


(* revision history
hm	29. sep 2007	rev 1.0
	original version

hm	5. oct 2007		rev 1.1
	added enable input

hm	6. oct 2007		rev 1.2
	added pos and angle inputs and outputs
	night position and angle can now be configured
	any manual operation at night will cancel night operation

*)
END_FUNCTION_BLOCK

(* POU sun_time, ST *)
FUNCTION_BLOCK sun_time
VAR_INPUT
	latitude : REAL;				(* latitude of geographical position  *)
	longitude : REAL;				(* longitude of geographical position  *)
	utc : DT;						(*	world time				*)
END_VAR
VAR_OUTPUT
	sun_midday : TOD;			(*	astrological midday in hours when sun stand at south direction	*)
	sun_rise : TOD;				(*	sun rise for current day in local time *)
	sun_set : TOD;				(*	sun set for current day in local time *)
	sun_declination : REAL;		(*	sun declination at midday in degrees	*)
END_VAR
VAR
	T: INT;							(* day in the year   *)
	DK: REAL;						(* sun declination at midday *)
	delta: REAL;					(* delta from midday for sunrise and sunset  *)
	h: REAL;
	B: REAL;
	offset : REAL;
END_VAR

(*
version 1.2	17 apr 2007
programmer 	hugo
tested by		tobias

this FUNCTION block calculates the sun rise, sun set, sun offset at midday sun declination for a given date 
for performance reasons the algorithm has been simplified and is accurate within a few minutes only 
the times are calculated in utc and have to be corrected for the given time zone
this correction is not done within sun_time because it would be a problem on days where dst is enabled or disabled

execution time on wago 750-841 is 30 us     
*)
B := Rad(latitude);
h := -0.0145;
T := day_of_year(DT_TO_DATE(utc));
offset := -0.1752 * SIN(0.033430*T + 0.5474) - 0.1340*SIN(0.018234*T - 0.1939);
sun_midday := hour_to_tod(12+Offset - longitude/15);
DK := 0.40954 * SIN(0.0172 * (T-79.35));
sun_declination := deg(DK);
delta := 12*ACOS((SIN(h) - SIN(B) * SIN(DK)) / (COS(B) * COS(DK)))/PI;
sun_rise := hour_to_tod(12 - delta - offset - longitude/15);
sun_set := hour_to_tod(12 + delta - Offset - longitude/15);

(* revision history

rev 1.1	hm	20.1.2007
	deleted unused variables sun_rineR and sun_setR

rev 1.2 hm 17.4.2007
	corrected error while sun:midday would not be corrected for longitude.
*)
END_FUNCTION_BLOCK

(* POU rmp_test, CFC *)
PROGRAM rmp_test
VAR
	set, rst, en, ud : BOOL;
	y : BYTE;
	bsy, on, off : BOOL;
	y1 : WORD;
	bsy1, on1, off1 : BOOL;
	x1: rmp_B;
	x2 : rmp_W;
	x3 : rmp_W;
	x6: RS;
	x4: TP;
	x5: TP;
	ramp: BYTE;
	x7: rmp_B;
	rmp1: BYTE;
	rmp2: BYTE;
	bsy2: BOOL;
	bsy0: BOOL;
	ramp0: WORD;
	x8: m_t;
	tt: TIME;
	x9: m_t;
	t1: TIME;
	x10: m_t;
	t2: TIME;
END_VAR
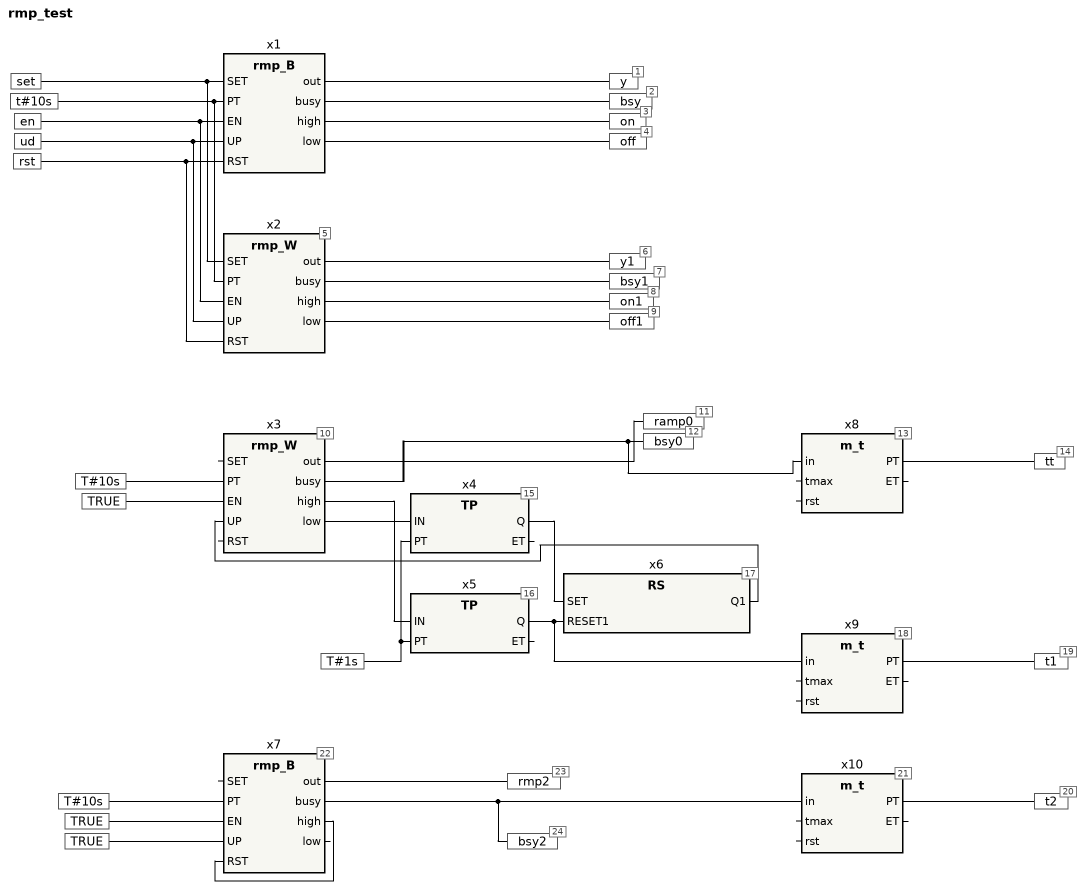
_CFC_ (* Continuous Function Chart, elements in execution order *)
#0 x1:rmp_B(SET: set, PT: t#10s, EN: en, UP: ud, RST: rst)
#1 y <= #0.out
#2 bsy <= #0.busy
#3 on <= #0.high
#4 off <= #0.low
#5 x2:rmp_W(SET: set, PT: t#10s, EN: en, UP: ud, RST: rst)
#6 y1 <= #5.out
#7 bsy1 <= #5.busy
#8 on1 <= #5.high
#9 off1 <= #5.low
#10 x3:rmp_W(SET: -, PT: T#10s, EN: TRUE, UP: #17.Q1, RST: -)
#11 ramp0 <= #10.out
#12 bsy0 <= #10.busy
#13 x8:m_t(in: #10.busy, tmax: -, rst: -)
#14 tt <= #13.PT
#15 x4:TP(IN: #10.low, PT: T#1s)
#16 x5:TP(IN: #10.high, PT: T#1s)
#17 x6:RS(SET: #15.Q, RESET1: #16.Q)
#18 x9:m_t(in: #16.Q, tmax: -, rst: -)
#19 t1 <= #18.PT
#20 t2 <= #21.PT
#21 x10:m_t(in: #22.busy, tmax: -, rst: -)
#22 x7:rmp_B(SET: -, PT: T#10s, EN: TRUE, UP: TRUE, RST: #22.high)
#23 rmp2 <= #22.out
#24 bsy2 <= #22.busy
_END_CFC_
(* the same logic as Structured Text *)
x1(SET := set, PT := t#10s, EN := en, UP := ud, RST := rst);
y := x1.out;
bsy := x1.busy;
on := x1.high;
off := x1.low;
x2(SET := set, PT := t#10s, EN := en, UP := ud, RST := rst);
y1 := x2.out;
bsy1 := x2.busy;
on1 := x2.high;
off1 := x2.low;
x3(PT := T#10s, EN := TRUE, UP := x6.Q1);
ramp0 := x3.out;
bsy0 := x3.busy;
x8(in := x3.busy);
tt := x8.PT;
x4(IN := x3.low, PT := T#1s);
x5(IN := x3.high, PT := T#1s);
x6(SET := x4.Q, RESET1 := x5.Q);
x9(in := x5.Q);
t1 := x9.PT;
t2 := x10.PT;
x10(in := x7.busy);
x7(PT := T#10s, EN := TRUE, UP := TRUE, RST := x7.high);
rmp2 := x7.out;
bsy2 := x7.busy;
END_PROGRAM

(* POU rmp_W, ST *)
FUNCTION_BLOCK rmp_W
VAR_INPUT
	SET : BOOL := FALSE;
	PT : TIME;
	EN : BOOL := TRUE;
	UP : BOOL := TRUE;
	RST : BOOL := FALSE;
END_VAR
VAR_OUTPUT
	out : WORD;
	busy : BOOL;
	high : BOOL;
	low : BOOL;
END_VAR
VAR
	last_step : DWORD;
	now : DWORD;
	tmp: DWORD;
	edge: BOOL;
	N: WORD;
END_VAR

(*
	version 1.5	5. oct 2007
	programmer 	oscat
	tested BY		oscat

this ramp generator generates a Word wide ramp with 65535 steps
the generator has an asynchronous set and reset
the ramp is controlled by PT which is the total ramp time for a full sweep from 0..65535
an UD input controlls the direction Up or Down and the E input enables the ramp generation
a busy output indicates that the ramp is running, busy false means output is stable.
the outputs low and high will be true when the output has reached its max or min value.
*)
(* read system time *)
now := T_PLC_US();

(* calculate the necessary step response *)
IF pt = t#0s THEN
	tmp := 65535;
ELSE
	tmp := SHL(now - last_step, 8) / (TIME_TO_DWORD(pt)*1000);
END_IF;
IF tmp > 65535 THEN N:= 65535; ELSE N:= DWORD_TO_BYTE(tmp); END_IF;

(* detetct edge on en *)
IF en AND NOT edge THEN
	last_step := now;
(* check for asynchronous set or reset *)
ELSIF rst THEN
	out := 0;
ELSIF set  THEN
	out := 65535;
ELSIF en AND N > 0 THEN
	(* generate ramp *)
	last_step := last_step + SHR(N * TIME_TO_DWORD(pt) * 1000,16);
	IF UP THEN
		IF out > 65535 - N THEN out := 65535; ELSE out := out + N; END_IF;
	ELSE
		IF out < N THEN out := 0; ELSE out := out - N; END_IF;
	END_IF;
END_IF;
edge := en;

(* checks for outputs stable and reset or set busy flag *)
IF out = 0 THEN
	busy := FALSE;
	low := TRUE;
	high := FALSE;
ELSIF out = 65535 THEN
	busy := FALSE;
	high := TRUE;
	low := FALSE;
ELSE
	busy := en;
	high := FALSE;
	low := FALSE;
END_IF;

(* revision history:

hm 4.10.2006		rev 1.1
	added the busy output which signals that the ramp is running.

hm 22.1.2007		rev 1.2
	deleted unused variable step

hm	17.9.2007		rev 1.3
	replaced time() with t_plc_ms() for compatibility reasons

hm	28. sep 2007	rev 1.4
	added outputs on and off
	busy is now disabled while en is false
	new coding for higher accuracy and performance

hm	5. oct 2007		rev 1.5
	added statements to allow for PT to be t#0s output jumps to max or min immediately

*)
END_FUNCTION_BLOCK

(* POU m_t, ST *)
FUNCTION_BLOCK m_t
VAR_INPUT
	in: BOOL;
	tmax : TIME := t#10d;
	rst: BOOL;
END_VAR
VAR_OUTPUT
	PT : TIME := t#0ms;
	ET: TIME;
END_VAR
VAR
	edge : BOOL := 0;
	start : TIME;
	stop : TIME;
	init : BOOL;
	tx: TIME;
	startup: BOOL;
END_VAR

(*
	version 1.2	16 sep 2007
	programmer 	hugo
	tested BY		tobias

m_t measures the with of a high pulse and returs the last measured pulse width on output PT.
a second output ET is starting from 0 at the rising edge and counting up until the falling edge occurs and resetts et to 0.
the asynchrtonous input rst can reset the outputs at any time.
tmax defines a maximum measurable time, if this value is exceeded the outputs will be reset to 0.
*)
(* check for rst input *)
IF rst OR et >= tmax THEN
	init := FALSE;
	startup := FALSE;
	pt := t#0ms;
	et := t#0ms;
END_IF;

(* avoid timers to start when input is true at startup *)
IF NOT startup THEN
	edge := in;
	startup := TRUE;
END_IF;

(* read system timer *)
tx := DWORD_TO_TIME(T_PLC_MS());

(* edge trigger rising and falling edge *)
IF in XOR edge THEN
	edge := in;
	(* rising edge starts measurement *)
	IF in THEN
		init := TRUE;
		start := Tx;
	(* falling edge stops measurement *)
	ELSIF init THEN
		stop := Tx;
		pt := stop - start;
	END_IF;
END_IF;

IF init AND in THEN
	et := Tx - start; ELSE et := t#0ms;
END_IF;

(* revision history
hm		4.8.2006	rev 1.0
	original version

hm		2.5.2007	rev 1.1
	added init variable to avoid unreasonable measurement if falling edge occurs first.
	added et (elapsed time) output to count from 0 at rising edge until a falling edge resets et to 0.
	added reset input.

hm		16.9.2007	rev 1.2
	changes time() to T_plc_ms() for compatibility reasons

*)
END_FUNCTION_BLOCK

(* POU actuator_2P, ST *)
FUNCTION_BLOCK actuator_2P
VAR_INPUT
	val : REAL;
	force : BOOL;
	force_in : BOOL;
END_VAR
VAR_INPUT CONSTANT
	self_act_time : TIME := t#10d;
	self_act_cycles : INT := 5;
	cycle_time : TIME := t#10m;
	min_ontime : TIME := t#10s;
	min_offtime : TIME := t#10s;
END_VAR
VAR_OUTPUT
	out :BOOL;
	pos : REAL;
END_VAR
VAR
	last_activation : TIME;
	count : INT;
	TON : TIME;
	tx : TIME;
	tc : TIME;
END_VAR


(*
version 1.3	15 sep 2007
programmer 	hugo
tested by		tobias

this is an intelligent actuator interface for any 2point actuator like coil drive.
the 2Point actuator can only switch on/off and therefore a input must be converted to on/off cycles.
the interface can be programmed with double click on the symbol for duty cyle, min_ontime and min_offtime to avoid flickering of the valve or flap.
in addition a self_act_time and self_act_cycles ca be programmed to switch n times on/off every self_act_time to avoid a valve to freeze.
a on and off input can be used to force the valve on or off at all times.
a additional pos output will always indicate the current position of a valve.
the input value must be between 0 and 1.

val		force	force_in	pos	out			
X		0		-			X		duty cycle X
-		1		1			1		1
-		1		0			0		0

*)
(* read system Time *)
tx := DWORD_TO_TIME(T_PLC_MS());
tc := tx - last_activation;

(* verify input to be between 0 and 1 *)
IF val <0 THEN val := 0; ELSIF val > 1 THEN val := 1; END_IF;

(* check for min ontime or min offtime and wait if not passed *)
IF (out AND tc < min_ontime) OR (NOT out AND tc < min_offtime) THEN RETURN;

(* when force off then shutoff valve *)
ELSIF force AND NOT force_in THEN
	pos := 0;
	out := 0;
	last_activation := tx;
	count := 0;

(* if force on then turn on valve *)

ELSIF force AND force_in THEN
	pos := 1;
	out := 1;
	last_activation := tx;
	count := 0;

(* if nothing happened for self_act_time then do self activation cycles *)
ELSIF (tc >= self_act_time AND count = 0 AND self_act_cycles > 0) OR (count > 0 AND count < self_act_cycles * 2) THEN
	out := NOT out;
	last_activation := tx;
	count := count + 1;
	RETURN;
ELSIF count > 0 THEN
	count := 0;
ELSE
	ton := multime(cycle_time,val);
	IF ton < min_ontime / 2 THEN ton := t#0s; ELSIF ton < min_ontime THEN ton := min_ontime; END_IF;
	IF ton > cycle_time - min_offtime / 2 THEN ton := cycle_time; ELSIF ton > cycle_time - min_offtime THEN ton := cycle_time - min_offtime; END_IF;
	IF ton = t#0s THEN
		IF out =0 THEN
			pos := 0;
			RETURN;
		ELSE
			out := 0;
			pos := 0;
			last_activation := tx;
		END_IF;
	ELSIF ton = cycle_time THEN
		IF out = 1 THEN
			pos := 1;
			RETURN;
		ELSE
			out := 1;
			pos := 1;
			last_activation := tx;
		END_IF;
	END_IF;
	pos := TIME_TO_REAL(ton) / TIME_TO_REAL(cycle_time);
	(* output pulse generation *)
	IF out AND tc >= ton THEN
		out := 0;
		last_activation := TIME();
	ELSIF NOT out AND tc >= cycle_time - ton THEN
		out := 1;
		last_activation := tx;
	END_IF;
END_IF;


(*
revision history:

7.10.2006: rev 1.1
	changed error pos could not reach 1 or 0 under certain conditions due to error in code.
	changed on and off in force and force_in for better usability.

17.1.2007	rev 1.2
	deleted unused variable time_overflow

15.9.2007	hm	rev 1.3
	replaced time() with T_PLC_MS for compatibility and performance reasons
*)
END_FUNCTION_BLOCK

(* POU cycle_time, ST *)
FUNCTION_BLOCK cycle_time
VAR_INPUT
	rst : BOOL;
END_VAR
VAR_OUTPUT
	ct_min : TIME := t#0s;
	ct_max : TIME := t#0s;
	ct_last : TIME;
	systime : TIME;
	sysdays : INT;
	cycles : DWORD;
END_VAR
VAR
	last_cycle : TIME;
	tx: TIME;
	init: BOOL;
END_VAR


(*
	version 1.2	16 sep 2007
	programmer 	hugo
	tested BY		hans

this function block measures the cycle time and displays the last, min and max cycle time of the current task.
the resolution is 1ms.
the cycles output is a dword counter which counts the cycles.
a rst pulse on the input will reset all data.


*)
tx := DWORD_TO_TIME(T_PLC_MS()) - last_cycle;
IF rst THEN
	ct_min := t#10h;
	ct_max := t#0ms;
	cycles := 0;
ELSIF last_cycle > t#0s THEN
	IF tx < ct_min THEN ct_min := tx;
	ELSIF tx > ct_max THEN ct_max := tx;
	END_IF;
	ct_last := tx;
ELSIF ct_min = t#0s THEN
	ct_min := t#0s - t#1ms;
END_IF;
IF init THEN
	systime := systime + tx;
		IF systime >= t#1d THEN
			systime := systime - t#1d;
			sysdays := sysdays + 1;
		END_IF;
END_IF;
init := TRUE;
last_cycle := last_cycle + tx;
cycles := cycles + 1;

(*	revision history
hm 12.12.2006		rev 1.1
	added cycles output, a dword cycle counter.
hm 10.3.2007			rev 1.2
	changed initialization of ct_min to t#10h for compatibility with siemens s7

hm	16.9.2007		rev 1.2
	changed Time() in T_PLC_MS() for compatibility resons

*)
END_FUNCTION_BLOCK

(* POU actuator_3P, ST *)
FUNCTION_BLOCK actuator_3P
VAR_INPUT
	in : REAL;
	force : BOOL;
	on : BOOL;
	end_pos : BOOL;
	diag : BOOL;
END_VAR
VAR_INPUT CONSTANT
	min_ontime : TIME := t#10s;
	min_offtime : TIME := t#10s;
	max_runtime : TIME := t#60s;
	auto_diag_time : TIME := t#10d;
	cal_runtime : TIME := t#600s;
	switch_available: BOOL;
END_VAR
VAR_OUTPUT
	out1 : BOOL;
	out2 : BOOL;
	pos : REAL;
	busy : BOOL;
	error : BOOL;
END_VAR
VAR
	val: REAL;
	tx : TIME;
	last_diag: TIME;
	last : TIME;
	runtime_1 : TIME;
	runtime_2 : TIME;
	state : INT;
	rout: FT_rmp;
	end : R_TRIG;
	cal_timer: TIME;
	Tn: TIME;
END_VAR


(*
version 1.3	 15 sep 2007
programmer 	hugo
tested by		tobias

actuator_3P is an interface for a 3 point actuator.
a 3P actuator is a motor with 2 directions that drives a valve or flap. the position of the valve or flap is controlled by runtime of the motor foreward or backward.
the available inputs are:
in is a real value which specifies the position of the actuator, 0 = 0% and 1 = 100% any value <0 or > 1 is limited to 0 or 1.
a force input must be low for normal operation and if switched high, the motor can only be controlled for 0% or 100% positions with the on input.
an and pos input is available for a end_pos switch, this switch indicates the valve or flap to be at either 0% or 100%
a diag input can at any time start a diag cycle which turns the motor towards the 0% position, then measures the runtime to 100% and then the runtime to 0%
these runtimes are stored and used for absolute positioning of the motor during normal operation.
a setup constand "auto_diag_time can be used to specify how often the actuator repeates this auto_diag cycla automatically.
at power on a cycle is perfomed automatically.
a 0 for this value means auto diag is never performed.

the outputs ar out1 and out2 for up and down direction of the motor. to avoid flickering the output can be programmed for min_ontime and min_offtime.
a pos outout indicates the absulute position of the actuator during operation and a busy output indicates the actuator is busy.
a error output is initiated when the specified max_runtime is reached by any direction during debug.
also when the up and down direction differs by more then 10% the error output is set.

for absolute positioning accuracy the actuator has a setup variable "cal_runtime" if this is set the actuator measures the total runtime of the motors and when this 
cal_runtime is exceeded it resets the actuator to 0% position and sets the output again to assure absolute accuracy.

autodiag and calibration can be shut off by setting the appropriate values to 0.
a switch_available setup variable specifies if end_pos switches are available.

*)
(* setup *)
Tn := DWORD_TO_TIME(T_PLC_MS());
tx := Tn - last;
end(clk := end_pos);

(* init only when first started *)
IF state = 0 THEN
	runtime_1 := max_runtime;
	runtime_2 := max_runtime;
	state := 1;
	rout(KR := 1000 / TIME_TO_REAL(runtime_1), KF := 1000 / TIME_TO_REAL(runtime_1) );
	tx := t#0s;
	last := Tn;
	last_diag := last;
END_IF;

(* check for end_sw and stop if reached *)
IF switch_available AND out1 AND end.Q THEN
	(* upper limit has been reached *)
	out1 := 0;
	rout(rmp := 0, in := 1);
	rout.Rmp := 1;
ELSIF switch_available AND out2 AND end.Q THEN
	(* lower limit has been reached *)
	out2 := 0;
	rout(rmp := 0, in := 0);
	rout.Rmp := 1;
END_IF;

(* check for min_offtime and min_ontime and return if it has not elapsed *)
IF NOT busy AND tx < min_offtime THEN RETURN;
ELSIF busy AND tx < min_ontime THEN RETURN;

(* check for last diag cycle and start diag if auto_diag_time has elapsed *)
ELSIF (tn - last_diag > auto_diag_time AND state > 10 AND auto_diag_time > t#0s) OR (diag AND state >= 10) THEN state := 1;

(* check if force pin is high *)
ELSIF force THEN state := 10;

(* check if calibration is necessary *)
ELSIF cal_timer > cal_runtime AND state = 99 AND cal_runtime > t#0s THEN state := 20;
END_IF;

(* state machine for operation *)
CASE state OF

1 :	(* diagnostic start *)
	(* all data is reset and out2 is turned on to make sure we start from top position *)
	last_diag := tn;
	diag := 0;
	state := 2;
	pos := 0;
	busy := 1;
	last := tn;
	out1 := 0;
	out2 := 1;
	RETURN;

2:	(* wait for max_runtime or end_pos to be reached *)
	IF tx < max_runtime AND NOT end.Q THEN RETURN; END_IF;
	state := 3;
	last := tn;
	out1 := 1;
	out2 := 0;
	RETURN;

3: 	(* measure runtime_2 *)
	IF tx < max_runtime AND NOT end.Q THEN RETURN; END_IF;
	state := 4;
	runtime_1 := tx;
	last := tn;
	out1 := 0;
	out2 := 1;
	RETURN;

4:	(* measure runtime_1 *)
	IF tx < max_runtime AND NOT end.Q THEN RETURN; END_IF;
	state := 99;
	runtime_2 := tx;
	last := tn;
	out2 := 0;
	busy := 0;
	(* reset the output ramp generator to the 0% position as the valve is after diags *)
	rout(rmp := 0, in := 0);
	rout.Rmp := 1;
	cal_timer := t#0s;
	IF differ(TIME_TO_REAL(runtime_1), TIME_TO_REAL(runtime_2), TIME_TO_REAL(max_runtime) * 0.1) THEN error := TRUE;
	ELSIF runtime_1 > multime(max_runtime, 0.9) AND switch_available THEN error := TRUE;
	ELSIF runtime_2 > multime(max_runtime, 0.9) AND switch_available THEN error := TRUE;
	END_IF;
	RETURN;

10: (* force pin is active, outputs are forced on or off by the on pin *)
	IF on AND NOT out2 THEN val := 1;
	ELSIF NOT on AND NOT out1 THEN val := 0;
	END_IF;
	IF NOT force THEN state := 99; END_IF;

20 : (* calibrate to allow for correction of positioning error addig up *)
	cal_timer := t#0s;
	state := 21;
	pos := 0;
	busy := 1;
	last := tn;
	out1 := 0;
	out2 := 1;
	RETURN;

21:	(* after end_sw or max_runtime we can be sure to have reached the 0% position *)
	IF tx < max_runtime AND NOT end.Q THEN RETURN; END_IF;
	state := 99;
	out2 := 0;
	busy := 0;
	last := tn;
	rout(rmp := 0, in := 0);
	rout.Rmp := 1;
	RETURN;

99: (* normal operation *)
	(* only if input changes for an equivalent of min_ontime then change the output *)
	(* if there is a directional change then wait until last step is finished *)
	IF in < TIME_TO_REAL(min_ontime)/TIME_TO_REAL(max_runtime)/2 THEN val := 0;
	ELSIF in > 1 - TIME_TO_REAL(min_ontime)/TIME_TO_REAL(max_runtime)/2 THEN val := 1;
	ELSIF differ(LIMIT(0,in,1), val, TIME_TO_REAL(min_ontime) / TIME_TO_REAL(max_runtime)) OR in = 0 OR in = 1 THEN
		IF in < val AND NOT out1 THEN val := in;
		ELSIF in > val AND NOT out2 THEN val := in;
		END_IF;
	END_IF;

END_CASE;

(* output ramp generator *)
rout(in := val);
out1 := rout.busy AND rout.UD;
out2 := rout.busy AND NOT rout.UD;
pos := rout.out;

(* set the busy output and if busy goes low, then set the last time in order to check for min_offtime *)
IF NOT busy AND rout.busy THEN
	last := tn;
ELSIF busy AND NOT rout.busy THEN
	cal_timer := cal_timer + tx;
	last := tn;
END_IF;
busy := rout.busy;



(* revision history

19.10.2006	rev 1.1
	added security checks for end_switch to avoid overrun of the end_switch, hans

23.1.2007		rev 1.2
	deleted unused variables force_on and force_off

15.9.2007	hm	rev 1.3
	replaced Time() with T_PLC_MS for compatibility and performance reasons

*)
END_FUNCTION_BLOCK

(* POU actuator_pump, ST *)
FUNCTION_BLOCK actuator_pump
VAR_INPUT
	in : BOOL;
	manual : BOOL;
	rst : BOOL := FALSE;
END_VAR
VAR_INPUT CONSTANT
	min_ontime : TIME := t#10s;
	min_offtime : TIME := t#10s;
	run_every : TIME := t#10000m;
END_VAR
VAR_OUTPUT
	pump : BOOL;
	runtime : REAL;
	cycles : REAL;
END_VAR
VAR
	tx : TIME;
	last_change : TIME;
	meter : ontime;
	old_man : BOOL;
	init: BOOL;
END_VAR

(*
	version 1.2	15 sep 2007
	programmer 	oscat
	tested BY		oscat

actuator_pump is a pump interface which can be controlled by an input in and an input manual.
in or manual high turns the pump output on.
a rst input is used to reset the runtime counters.
when the pump was not active for a time run_every the actuator turns on the pump automatically for min_ontime.
two setup variables min_ontime and min_offtime guarantee a minimum runtime and offtime of the pump.
the units are hours and the output type is real to prevent from overfow.

*)
tx := DWORD_TO_TIME(T_PLC_MS());

IF NOT init THEN
	init := 1;
	last_change := tx;
ELSIF rst THEN
	rst := FALSE;
	meter(rst := 1);
	meter.rst := 0;
ELSIF manual AND NOT pump AND NOT old_man THEN
	last_change := tx;
	pump := 1;
ELSIF NOT manual AND old_man AND pump AND NOT in THEN
	last_change := tx;
	pump := 0;
ELSIF in AND NOT pump AND tx - last_change >= min_offtime THEN
	last_change := tx;
	pump := 1;
ELSIF pump AND NOT in AND NOT manual AND tx - last_change >= min_ontime THEN
	last_change := tx;
	pump := 0;
ELSIF NOT pump AND tx - last_change >= run_every THEN
	last_change := tx;
	pump := 1;
END_IF;

meter(in := pump);
runtime := meter.ontime;
cycles := meter.cycles;
old_man := manual;

(*
27.12.2006	rev 1.1	hm
	fixed a failure while the pump would run for tmin after startup.

15.9.2007	hm	rev 1.2
	replaced Time() with T_PLC_MS for compatibility and performance reasons

*)
END_FUNCTION_BLOCK

(* POU Meter, ST *)
FUNCTION_BLOCK Meter
VAR_INPUT
	M1, M2 : REAL;
	I1, I2 : BOOL;
	D : REAL := 1;
	RST : BOOL;
END_VAR
VAR_OUTPUT RETAIN
	MX : REAL;
END_VAR
VAR
	int1 : FT_INT;
	int2 : FT_INT;
END_VAR

(*
	version 1.0	16 sep 2007
	programmer 	oscat
	tested BY		oscat

METER measures usage of power or similar values the output MX is the summ of the inputs over time.
MX := sum over time of I1 * P1 + I2 * P2.
a simple example is the consumption counter for a 2 stage oil burner where stage 1 is 10KW and stage 2 is 20KW.
I1 and I2 decide which value is accounted for, I1 = True only counts P1, I2 is True counts P2 
and I1 and I2 is true counts P1 and P2.
the meter can be used for all kind of consumption meters. P1 and P2 can change on the fly.

*)
int1(in := M1, Run := I1, RST := RST, out_min := -1E-38, out_max :=3E+38);
int2(in := M2, Run := I2, RST := RST, out_min := -1E-38, out_max :=3E+38);
MX := (int1.Out + int2.Out) / D;

(* revision history

hm	7.2.2007		rev 1.0
	original version

*)
END_FUNCTION_BLOCK

(* POU FT_INT, ST *)
FUNCTION_BLOCK FT_INT
VAR_INPUT
	in : REAL;
	K : REAL := 1;
	run : BOOL := 1;
	rst: BOOL := 0;
	out_min : REAL := -1000;
	out_max : REAL := 1000;
END_VAR
VAR_OUTPUT
	Out : REAL;
	ET: TIME;
END_VAR
VAR
	last: DWORD;
	in_last : REAL;
	tx: DWORD;
	init: BOOL;
	tc: DWORD;
	eti : DWORD;
END_VAR


(*
version 1.3	15 sep 2007
programmer 	hugo
tested by		tobias

FT_int is an integrator with input IN and factor K.
integration is only done while run = true, if run is false integration is stopped and the out remains at the last value.
if run is left unconnected, run is considered true by the function block.
the output ET will display the total integration time from last reset.
a rst input will reset output and the timer ET to 0.
the out_min and out_max values can be set to ,imit the output value range. 
out _min is preset to -1000 and out_max is preset to 1000.
the default for K is 1.

 
*)
(* read and store system time *)

last := tx;
tx := T_PLC_US();
tc := tx - last;

(* startup initialisation *)
IF rst OR NOT init THEN
	out := 0;
	ET := t#0s;
	init := TRUE;
	last := tx;
ELSIF run THEN
	out := out + (in + in_last)/2 * tc * K / 1000000;
	IF out < out_min THEN out := out_min; ELSIF out > out_max THEN out := out_max; END_IF;
	eti := eti + tc;
	et := DWORD_TO_TIME(eti / 1000);
END_IF;
in_last := in;

(*
hm 13.12.2006	rev 1.1
	changed to "trapezregel" which increases accuracy
	before out := out + in * time new: out := out + (in + in_last) / 2 * time

hm 15.1.2007		rev 1.2
	added default for k to be 1.

hm	15.9.2007		rev 1.3
	replaced time() with T_PLC_US for compatibility and performance reason
	increased internal accuracy to microseconds
*)
END_FUNCTION_BLOCK

(* POU ontime, ST *)
FUNCTION_BLOCK ontime
VAR_INPUT
	in : BOOL;
	rst : BOOL := FALSE;
END_VAR
VAR_OUTPUT RETAIN
	ontime : REAL;
	last_on : REAL;
	cycles : REAL;
END_VAR
VAR
	tx: DWORD;
	last : DWORD;
	edge : BOOL := 0;
	L_time1, H_time1, L_time2, H_time2 : DWORD;
	temp: DWORD;
END_VAR

(*
version 1.3	16 sep 2007
programmer 	oscat
tested by		tobias

M_runtime measures the ontime of a signal in hours.
the output is of type real because the time type will overflow within 49 days.
the units are hours.

*)
(* read system time *)
tx := T_PLC_MS();

IF rst THEN
	L_time1 := 0;
	H_time1 := 0;
	cycles := 0;
	L_time2 := 0;
	H_time2 := 0;
	ontime := 0;
	last_on := 0;
ELSIF in THEN
	temp := L_time1;
	L_time1 := L_time1 + (tx-last);
	IF temp > L_time1 THEN H_time1 := H_time1 + 1; END_IF;
	ontime := L_time1/3600000.0 + EXPT(2,32)/3600000.0 * H_time1;
	temp := L_time2;
	L_time2 := L_time2 + (tx-last);
	IF temp > L_time2 THEN H_time2 := H_time2 +2; END_IF;
	last_on := L_time2/3600000.0 + EXPT(2,32)/3600000.0 * H_time2;
	IF NOT edge THEN
		cycles := cycles +1;
		last_on := 0;
		L_time2 := 0;
		H_time2 := 0;
	END_IF;
END_IF;
last := tx;
edge := in;

(* revision history
hm 22.2.2007		rev 1.1
	changed VAR RETAIN PERSISTENT to VAR RETAIN for better compatibility
	wago lon contollers do not support persisitent

hm 2.8.2007		rev 1.2
	adding time up in a real number will automatically lead to the point where 
	small time scales like the cycle time will be below the resolution of real and therefore
	ontime would not increase in small steps as necessary
	the time is now measured internally in two  dwords and be converted to real only for
	output purposes.
	deleted the variable power because it was unnecessary

hm	16.9.2007	rev 1.3
	changes time() to T_plc_ms() for compatibility reasons

*)
END_FUNCTION_BLOCK

(* POU actuator_UD, ST *)
FUNCTION_BLOCK actuator_UD
VAR_INPUT
	UD : BOOL;
	ON : BOOL;
	Manual : BOOL := 0;
	Up : BOOL;
	Dn : BOOL;
	off : BOOL := 0;
	YUP_in : BOOL;
	YDN_in : BOOL;
END_VAR
VAR_INPUT CONSTANT
	TON : TIME;
	TOFF : TIME;
	out_return : BOOL;
END_VAR
VAR_OUTPUT
	Yup : BOOL;
	Ydn : BOOL;
	status : BYTE;
END_VAR
VAR
	tx : TIME;
	last : TIME;
	init: BOOL;
END_VAR

(*
version 1.2	15 sep 2007
programmer 	hugo
tested by		tobias

out_ud is a up/dn or Right/left locked output driver.
it can be controlled by automatic inputs UD and ON as well as manual inputs for up and dn.
a security input to shut off at any time is prvided by the off input.
two time set inputs ton and toff specify a minimum on time for outputs and a minimum off time before the next output can become active.
the module assures that only one output can be active at any time.
for higher security pls make sure you use hardware locking of the outputs to prevent from defective wiring or outputs.
further security is provided b feedback inputs Yup_in and Ydn_in which are separate inputs for the output signal, if these inputs are not available 
pls connect them directly to Yup and Ydn.
manual mode will override automatic mode by setting the manual input high.
a status output will be 0 for normal operation or 1 - 99 for error reporting and 101 - 199 for status reporting
The status output is ESR comptible.
*)
(* read system time *)
tx := DWORD_TO_TIME(T_PLC_MS());

IF NOT init THEN
	(* INITIALIZATION AT FIRST CALL *)
	last := tx;
	init := TRUE;
ELSIF off THEN
	(* emergency shut off detected *)
	Yup := FALSE;
	Ydn := FALSE;
	last := tx;
	status := 101;

(* WATH FOR MIN TON TIME *)
ELSIF ((Yup OR Ydn) AND tx - last < Ton) THEN RETURN;
ELSIF NOT yup AND NOT ydn AND tx - last < toff THEN	RETURN;

(* manual operation *)
ELSIF manual THEN
	status := 102;
	(* directional chage set both outs 0 first *)
	IF yup AND NOT up OR ydn AND NOT dn THEN
		ydn := 0;
		yup := 0;
		last := tx;
	(* manual up operation *)
	ELSIF UP AND NOT DN AND NOT OFF THEN
		Ydn := 0;
		Yup := 1;
		last := tx;
		status := 103;
	(* manual down operation *)
	ELSIF DN AND NOT UP AND NOT OFF THEN
		Yup := 0;
		Ydn := 1;
		last := tx;
		status := 104;
	(* maual mode but no up or down *)
	ELSE
		IF YUP OR YDN THEN LAST := tx; END_IF;
		Yup := 0;
		Ydn := 0;
	END_IF;

(* automatic operation *)
ELSE
	(* directional change set outputs low first *)
	IF yup AND NOT ud OR ydn AND UD THEN
		yup := 0;
		ydn := 0;
		last := tx;
	(* automatic up operation *)
	ELSIF Ud AND on AND NOT OFF THEN
		Ydn := 0;
		Yup := 1;
		last := tx;
		status := 111;

	(* automatic down operation *)
	ELSIF NOT UD AND on AND NOT OFF THEN
		Yup := 0;
		Ydn := 1;
		last := tx;
		status := 112;
	(* standby mode *)
	ELSE
		IF Yup OR Ydn THEN last := tx; END_IF;
		Yup := 0;
		Ydn := 0;
		status := 110;
	END_IF;
END_IF;

(* make sure Yup and Ydn are never on at the same time *)
IF Ydn AND Yup_in AND out_return THEN
	Ydn := 0;
	status := 1;
END_IF;
IF Yup AND Ydn_in AND out_return THEN
	Yup := 0;
	status := 2;
END_IF;

(* revision history
hm 22. jan 2007	rev 1.1
	added status output
	changed inputs ton, toff to config variables
	added config var out_return to enable yup_in and Ydn_in
	manual mod will override automatic mode 

hm	15.9.2007	rev 1.2
	replaced Time() with T_PLC_MS for compatibility and performance reasons
*)
END_FUNCTION_BLOCK

(* POU astro, ST *)
FUNCTION_BLOCK astro
VAR_INPUT
	m : REAL;
	AE : REAL;
	PC : REAL;
	LJ : REAL;
END_VAR
VAR_OUTPUT
	Ym : REAL;
	YAE : REAL;
	YPC : REAL;
	YLJ : REAL;
END_VAR
VAR
END_VAR

(*
version 1.0	27 mar 2007
programmer 	hugo
tested by		oscat

this function converts different length units
any unused input can simply be left open.
different inputs connected at the same time will be added up.

*)
YAE :=	AE
		+ m / 149.597870E9
		+ PC * 206265
		+ LJ * 63240;
Ym := YAE * 149.597870E9;
YPC := YAE / 206265;
YLJ := YAE / 63240;


(*
Länge Meter m SI-Basiseinheit
Astronomische Einheit* AE 1 AE = 149,597 870 · E9 m
Parsec pc 1 pc = 206265 AE = 30,857 · E15 m
Lichtjahr Lj 1 Lj = 9,460 530 · E15 m = 63240 AE = 0,306 59 pc
Ångström Å 1 Å = E–l0 m
typograph. Punkt p 1 p = 0,376 065 mm • im Druckereigewerbe
inch** in 1 in = 2,54 · E–2 m = 25,4 mm***
foot ft 1 ft = 0,3048 m = 30,48 cm
yard yd 1 yd = 0,9144 m
mile mile 1 mile = 1609,344 m
Internat. Seemeile sm 1 sm = 1852 m
Fathom fm 1 fm = 1,829 m • in der Seeschifffahrt

*)
END_FUNCTION_BLOCK

(* POU B_TRIG, ST *)
FUNCTION_BLOCK B_TRIG
VAR_INPUT
	CLK : BOOL;
END_VAR
VAR_OUTPUT
	Q : BOOL := 0;
END_VAR
VAR
	edge : BOOL := 0;
END_VAR

(*
version 1.0	4 aug 2006
programmer 	hugo
tested by		tobias

this block is similar to R_trig and F_trig but it generates a pulse on rising and falling edge.

executioin TIME on wago 750-841 = 5us
*)
Q := clk XOR edge;
edge := CLK;
END_FUNCTION_BLOCK

(* POU bar_graph, ST *)
FUNCTION_BLOCK bar_graph
VAR_INPUT
	X : REAL;
	rst : BOOL;
END_VAR
VAR_INPUT CONSTANT
	trigger_Low : REAL;
	trigger_High : REAL;
	Alarm_low : BOOL;
	Alarm_high : BOOL;
	log_scale : BOOL;
END_VAR
VAR_OUTPUT
	LOW, Q1, Q2, Q3, Q4, Q5, Q6, HIGH : BOOL;
	Alarm : BOOL;
	Status : BYTE;
END_VAR
VAR
	init : BOOL;
	T1, T2, T3, T4, T5 : REAL;
END_VAR
VAR_TEMP
	temp : REAL;
END_VAR

(*
	version 1.0	22 feb 2007
	programmer 	hugo
	tested BY		hans

bar graph is a muti window comparator which displays an analog input signal on 8 digital outputs.
only one output is active a any given time depending on the value of the input signal.
the output can be of linear or logarithmic scale.

*)
IF NOT init THEN
	init := TRUE;
	IF log_scale THEN
		temp := EXPT(Trigger_high / Trigger_low, 1 / 6);
		T1 := trigger_low * temp;
		T2 := T1 * temp;
		T3 := T2 * temp;
		T4 := T3 * temp;
		T5 := T4 * temp;
	ELSE
		temp := (trigger_high - trigger_low) / 7;
		T1 := trigger_low + temp;
		T2 := T1 + temp;
		T3 := T2 + temp;
		T4 := T3 + temp;
		T5 := T4 + temp;
	END_IF;
END_IF;

(* clear outputs before checking *)
Q1 := FALSE;
Q2 := FALSE;
Q3 := FALSE;
Q4 := FALSE;
Q5 := FALSE;
Q6 := FALSE;
status := 110;

(* low, high and alarm can only be cleared with rst depending on alarm_low and alarm_high *)
IF NOT alarm_low THEN low := FALSE; END_IF;
IF NOT alarm_high THEN high := FALSE; END_IF;
IF rst THEN
	alarm := FALSE;
	low := FALSE;
	high := FALSE;
END_IF;

(* check and set outputs *)
IF X < trigger_low THEN
	Low := TRUE;
	status := 111;
	IF alarm_low THEN
		alarm := TRUE;
		status := 1;
	END_IF;
ELSIF X < T1 THEN
	Q1 := TRUE;
ELSIF x < t2 THEN
	Q2 := TRUE;
ELSIF x < t3 THEN
	Q3 := TRUE;
ELSIF x < T4 THEN
	Q4 := TRUE;
ELSIF x < T5 THEN
	q5 := TRUE;
ELSIF x < trigger_high THEN
	q6 := TRUE;
ELSE
	high := TRUE;
	status := 112;
	IF alarm_high THEN
		alarm := TRUE;
		status := 2;
	END_IF;
END_IF;
END_FUNCTION_BLOCK

(* POU Boiler, ST *)
FUNCTION_BLOCK Boiler
VAR_INPUT
	T_upper : REAL;
	T_lower : REAL;
	Pressure : BOOL := TRUE;
	enable : BOOL := TRUE;
	Req_1 : BOOL;
	Req_2 : BOOL;
	Boost : BOOL;
END_VAR
VAR_INPUT CONSTANT
	t_upper_min : REAL := 50;
	t_upper_max : REAL := 60;
	T_lower_enable : BOOL;
	T_lower_max : REAL := 60;
	T_request_1 : REAL := 70;
	T_request_2 : REAL := 50;
	T_request_hys : REAL := 5;
	T_protect_high : REAL := 80;
	T_protect_low : REAL := 10;
END_VAR
VAR_OUTPUT
	Heat : BOOL;
	error : BOOL;
	status : BYTE;
END_VAR
VAR
	edge: BOOL;
	boost_mode: BOOL;
	flag_0 : BOOL;
	flag_1: BOOL;
	flag_2: BOOL;
END_VAR

(*
version 1.0	27 feb 2007
programmer 	hugo
tested by		tobias

this function block controls a hot water boiler. The Boiler can be equipped with two temperature sensors on top and bottom of the tank, T_LOWER_ENABLE must be set to True in this case.
alternatively can BOILER be configured for one (TOP) temperature sensor only (T_LOWER_ENABLE set to False).
A Pressure sensor is used to detect fresh water pressure and disable all heating if there is no water pressure. This input is dset to True by default, so if it is not used it can simply be left open.
A enable input enables the hot water heating while it is set to True. alternatively can a Ture on Req_1 or Req_2 start the heating to predefined temperatures during setup.
A low to high edge on the boost input will start heating imediately until T_upper_max is reached, it can be used to generate extra hot water when needed.

*)
(* read sensors and check for valid data *)
IF t_upper > t_protect_high THEN
	status := 1;
	heat := FALSE;
	error := TRUE;
ELSIF t_upper < t_protect_low THEN
	status := 2;
	heat := TRUE;
	error := TRUE;
ELSIF t_lower > T_protect_high AND t_lower_enable THEN
	status := 3;
	heat := FALSE;
	error := TRUE;
ELSIF t_lower < t_protect_low AND t_lower_enable THEN
	status := 4;
	heat := TRUE;
	error := TRUE;
ELSIF NOT pressure THEN
	status := 5;
	heat := FALSE;
	error := TRUE;
ELSIF req_1 OR req_2 OR enable OR boost THEN
	error := FALSE;

	(* determine if heat needs to be turned on *)
	IF boost AND NOT edge AND t_upper < t_upper_max THEN
		status := 101;
		heat := TRUE;
		boost_mode := TRUE;
	ELSIF enable AND t_upper < T_upper_min THEN
		status := 102;
		heat := TRUE;
	ELSIF req_1 AND t_upper < T_request_1 THEN
		status := 103;
		heat := TRUE;
	ELSIF req_2 AND t_upper < t_request_2 THEN
		status := 104;
		heat := TRUE;
	END_IF;

	(* determine the shut off temperature *)
	IF heat THEN
		IF (enable OR boost_mode) THEN
			flag_0 := TRUE;
			IF T_lower_enable AND T_lower > T_lower_max THEN
				flag_0 := FALSE;
				boost_mode := FALSE;
			ELSIF NOT T_lower_enable AND T_upper > T_upper_max THEN
				flag_0 := FALSE;
				boost_mode := FALSE;
			END_IF;
		ELSE
			flag_0 := FALSE;
		END_IF;
		IF req_1 AND T_upper > T_request_1 + T_request_hys THEN flag_1 := FALSE; ELSE flag_1 := req_1; END_IF;
		IF req_2 AND T_upper > T_request_2 + T_request_hys THEN flag_2 := FALSE; ELSE flag_2 := req_2; END_IF;

		(* shut off heat if no longer needed *)
		heat := flag_0 OR flag_1 OR flag_2;
		IF heat = FALSE THEN status := 100; END_IF;
	END_IF;
ELSE
	status := 100;
	heat := FALSE;
	error := FALSE;
END_IF;
edge := boost;
END_FUNCTION_BLOCK

(* POU pressure, ST *)
FUNCTION_BLOCK pressure
VAR_INPUT
	mws : REAL;
	torr : REAL;
	att : REAL;
	atm : REAL;
	pa : REAL;
	bar : REAL;
END_VAR
VAR_OUTPUT
	Ymws : REAL;
	Ytorr : REAL;
	Yatt : REAL;
	Yatm : REAL;
	Ypa : REAL;
	Ybar : REAL;
END_VAR
VAR
END_VAR

(*
version 1.0	27 mar 2007
programmer 	hugo
tested by		oscat

this function converts different pressure units
any unused input can simply be left open.
different inputs connected at the same time will be added up.
*)
Ybar := bar +
		pa / 100000 +
		0.980665 * att +
		1.01325 * atm +
		0.001333224 * torr +
		0.0980665 * mws;
Ymws := ybar / 0.0980665;
Ytorr := ybar / 0.001333224;
Yatt := ybar / 0.980665;
yatm := ybar / 1.01325;
Ypa := ybar * 100000;


(*
Druck, Pascal Pa 1 Pa = 1 N/m2 = 1 kg/(s2 �E m) . 0,75 �E 10.2 mmHg
mechanische 1 MPa = 1 N/mm2 . fur Festigkeitsangaben
Spannung Bar bar 1 bar = 105 Pa = 103 mbar = 105 kg/(s2 �E m)
Millimeter- mmHg 1 mmHg = 133,322 Pa = 1,333 22 mbar
Quecksilbersaule . nur in Heilkunde zulassig
physik. Atmosphare atm 1 atm = 1,013 25 bar
techn. Atmosphare at 1 at = 1 kp/cm2 = 0,980665 bar
Torr Torr 1 Torr = (101325/760) Pa = 1,333224 mbar
Meter-Wassersaule mWS 1 mWS = 9806,65 Pa = 98,0665 mbar
psi lbf/in2 1 lbf/in2 = 68,947 57 mbar = 6894,757 Pa

*)
END_FUNCTION_BLOCK

(* POU Burner, ST *)
FUNCTION_BLOCK Burner
VAR_INPUT
	in : BOOL;
	stage2 : BOOL;
	over_temp : BOOL;
	oil_temp : BOOL := TRUE;
	Flame : BOOL;
	rst : BOOL;
	rst_timer : BOOL;
END_VAR
VAR_INPUT CONSTANT
	pre_heat_time : TIME := t#5s;
	pre_vent_time : TIME := t#15s;
	pre_ignite_time : TIME := t#5s;
	post_ignite_time : TIME := t#25s;
	stage2_delay : TIME := t#10s;
	safety_time : TIME := t#5s;
	lockout_time : TIME := t#10s;
	multiple_ignition : BOOL := TRUE;
	KW1 : REAL;
	KW2 : REAL;
END_VAR
VAR_OUTPUT
	motor : BOOL;
	coil1 : BOOL;
	coil2 : BOOL;
	pre_heat: BOOL;
	ignite : BOOL;
	runtime1 : REAL;
	runtime2 : REAL;
	KWh : REAL;
	cycles : REAL;
	status : BYTE;
	fail : BOOL;
END_VAR
VAR
	state : BYTE;
	last : TIME;
	tx: TIME;
	last_change: TIME;
	timer1 : ontime;
	timer2 : ontime;
	oil_temp_last: BOOL;
END_VAR

(*
version 1.5	15 sep 2007
programmer 	oscat
tested by		tobias

burner ist eine Oel-Brenner_steuerung fuer nichtmodulierende Oelbrenner
die steuerung kann ueber setup werte programmiert werden und entsprechenden brennern angepasst werden.
die vorheizzeit ist die zeit die eine oelvorwaermung aufgeheizt wird bevor der motor gestartet wird.
der eingang oil_temp gibt an ob die oil_temp erreicht wurde, er ist default auf true und kann auch offen gelassen werden.
die vorbelueftungszeit ist die zeit die der luefter laeuft bevor die oelzufuhr freigegeben wird.
die vorzuendzeit iust diejenige zeit die die zuendung vor offnen des oelventiel gestartet wird.
nachzuendzeit ist die zeit die nach entzuendung der flamme noch gezuendet wird.
die sicherheitszeit ist die zeit nach der die oelzufuhr gesperrt wird wenn keine flamme entsteht.
nach ablauf der sicherheitszeit wird ein fehler flag gesetzt und kann erst nach der sperrzeit wieder durch einen reset geloescht werden.
waehrend der sperrzeit ist keine weitere zuendung oder einschalten moeglich.
das flag mehrfachzuendung gibt an ob eine erloschene flamme in betrieb automatisch wieder gezuendet werden soll.
der flammwaechster liegt auf eingang flamme, ein uebertemperaturschutz auf dem eingang over_temp
der betriebsstundenzaehler gibt die brennerstunden in stunden als real ausgabewer an.
der ausgang motor steuert den luefter / pumpenmotor, oil_ventil schaltet das oil ventil und zuendung schaltet die zuendung ein.

if output fail > 0 an error happened and the output has an error code:
0 :	no error
1 :	pre heating time expired and oil temp input is not true
2 :	flame monitor is active during preheating time
3 :	flame monitor active during pre_ventilation_time
4 :	no ignoition during safety time
5 :	no flame during operation
9 :	overtemp input is true

*)
(* read system time *)
tx := DWORD_TO_TIME(T_PLC_MS());

(* check rst input and overtemp *)
IF rst OR over_temp OR state = 0 THEN
	IF status > 0 AND tx - last_change >= lockout_time AND rst THEN
		status := 110;
		fail := FALSE;
		state := 1;
	ELSE
		(* normaler reset *)
		motor := FALSE;
		coil1 := FALSE;
		coil2 := FALSE;
		ignite := FALSE;
		pre_heat := FALSE;
		IF over_temp THEN
			status := 9;
			fail := TRUE;
		END_IF;
		last_change := tx;
		last := tx;
		state := 1;
	END_IF;
END_IF;

(* check for timer rst and rst timer if true *)
IF rst_timer THEN
	timer1( rst := TRUE);
	timer1.rst := FALSE;
	timer2(rst := TRUE);
	timer2.rst := FALSE;
END_IF;

(* quit here if an error is present *)
IF (status > 0 AND status < 100) OR rst THEN RETURN; END_IF;

(* start sequence *)
CASE state OF

1:	(* in signal starts oil pre heating *)
	IF in AND flame THEN
		state := 7;
		pre_heat := FALSE;
		status := 2;
		last_change := tx;
	ELSIF in THEN
		pre_heat := TRUE;
		state := 2;
		last_change := tx;
	END_IF;

2:	(* after pre_heating time start motor *)
	IF (tx- last_change >= pre_heat_time AND oil_temp) OR (oil_temp AND NOT oil_temp_last) THEN
		motor := TRUE;
		state := 3;
		last_change := tx;
	(* pre_heat_time ist abgelaufen und oil_temp ist nicht aktiv *)
	ELSIF tx - last_change >= pre_heat_time AND NOT oil_temp THEN
		state := 7;
		pre_heat := FALSE;
		status := 1;
		last_change := tx;
	(* flame monitor cannot be active at this time *)
	ELSIF flame THEN
		state := 7;
		pre_heat := FALSE;
		status := 2;
		last_change := tx;
	END_IF;

3:	(* abwarten bis zündung eingeschaltet werden kann *)
	IF tx - last_change >= pre_vent_time - pre_ignite_time THEN
		ignite := TRUE;
		state := 4;
		last_change := tx;
	(* flame monitor cannot be active at this time *)
	ELSIF flame THEN
		state := 7;
		pre_heat := FALSE;
		motor := FALSE;
		status := 3;
		last_change := tx;
	END_IF;

4:	(* warten bis oelzufuhr geoeffnet werden darf *)
	IF tx - last_change >= pre_ignite_time THEN
		coil1 := TRUE;
		state := 5;
		last_change := tx;
	END_IF;

5:	(* warten auf flammwaechter und falls noetig abschalten *)
	IF tx - last_change >= safety_time OR flame THEN
		IF NOT flame THEN
			(* notabschaltung da flammwaechster nicht angesprochen hat *)
			state := 7;
			motor := FALSE;
			coil1 := FALSE;
			pre_heat := FALSE;
			ignite := FALSE;
			status := 4;
			last_change := tx;
		ELSE
			state := 6;
			last_change := tx;
		END_IF;
	END_IF;

6:	(* brenner läuft, flammueberwachung und nach ablauf der nachigniteszeit ignite abschalten *)
	IF NOT flame AND NOT multiple_ignition THEN
		(* notabschaltung da flammwaechster keine flamme meldet *)
		state := 7;
		motor := FALSE;
		coil1 := FALSE;
		coil2 := FALSE;
		pre_heat := FALSE;
		ignite := FALSE;
		status := 5;
		last_change := tx;
	ELSIF NOT flame AND multiple_ignition THEN
		ignite := TRUE;
		state := 5;
		coil2 := FALSE;
		last_change := tx;
	ELSE
		IF tx - last_change >= post_ignite_time THEN
			(* post_ignite_time abgelaufen, ignite abschalten *)
			ignite := FALSE;
		END_IF;
		IF tx - last_change >= stage2_delay AND stage2 THEN
			coil2 := TRUE;
		ELSE
			coil2 := FALSE;
		END_IF;
	END_IF;
END_CASE;

(* abschaltung wenn kein eingangssignal *)
IF NOT in THEN
	state := 1;
	motor := FALSE;
	coil1 := FALSE;
	coil2 := FALSE;
	ignite := FALSE;
	pre_heat := FALSE;
	last_change := tx;
END_IF;

(* runtimezähler *)
timer1(in := flame AND in AND motor AND coil1 AND NOT coil2);
timer2(in := flame AND in AND motor AND coil1 AND coil2);
runtime1 := timer1.ontime;
runtime2 := timer2.ontime;
cycles := timer1.cycles;
KWH := runtime1 * KW1 + runtime2 * KW2;

(* zeit fuer naechsten aufruf merken *)
last := tx;

(* set fail output IF ERROR and Status  if normal operation *)

IF status > 0 AND status < 100 THEN
	fail := TRUE;
ELSE
	fail := FALSE;
	IF NOT in THEN
		status := 110;
	ELSIF flame AND in AND motor AND coil2 AND coil1 THEN
		status := 113;
	ELSIF flame AND in AND motor AND coil1 THEN
		status := 112;
	ELSE
		status := 111;
	END_IF;
END_IF;


(*
31.12.2006	hm		rev 1.1
	added pre_heat timing and output
	flame monitor before ignition will generate error on status output
	added output for KWh

31.12.2006	hm		rev 1.2
	added oil_temp_input

31.12.2006	hm		rev 1.3
	changed status output to be byte instead of bool

22.1.2007		hm		rev 1.4
	renamed fail output to status
	added output cycles
	corrected an error while pre_heat would be on when an error was present
	added coil2 output and stage2 input

15.9.2007		hm		rev 1.5
	replaced Time() with T_PLC_MS for compatibility and performance reasons

*)
END_FUNCTION_BLOCK

(* POU Byte_to_Bit, ST *)
FUNCTION_BLOCK Byte_to_Bit
VAR_INPUT
	IN: BYTE;
END_VAR
VAR_OUTPUT
	B0: BOOL;
	B1: BOOL;
	B2: BOOL;
	B3: BOOL;
	B4: BOOL;
	B5: BOOL;
	B6: BOOL;
	B7: BOOL;
END_VAR
VAR
END_VAR

(*
version 1.0	4 aug 2006
programmer 	hugo
tested by		tobias

this Function Block extracts the 8 Bits from a byte

executioin TIME on wago 750-841 = 13us
*)
B0 := IN.0;
B1 := IN.1;
B2 := IN.2;
B3 := IN.3;
B4 := IN.4;
B5 := IN.5;
B6 := IN.6;
B7 := IN.7;
END_FUNCTION_BLOCK

(* POU Calibrate, ST *)
FUNCTION_BLOCK Calibrate
VAR_INPUT
	X : REAL;
	CO : BOOL;
	CS : BOOL;
END_VAR
VAR_INPUT CONSTANT
	Y_Offset : REAL;
	Y_Scale : REAL;
END_VAR
VAR_OUTPUT
	Y : REAL;
END_VAR
VAR RETAIN
	offset : REAL;
	Scale : REAL := 1;
END_VAR

(*
	version 1.2	22 feb 2007
	programmer 	hugo
	tested BY		hans

Calibrate allows for offset and scale calibration of an analog input.
offset is calibrated to a stored reference Y_offset while CO is true.
after the offset is calibrated, scale can be calibrated to a reference value Y_scale while CS is true.
*)
(* check for calibration *)
IF CO THEN
	Offset := Y_Offset - X;
ELSIF CS THEN
	scale := Y_scale / (X+Offset);
END_IF;
(* calculate output *)
Y := (X + Offset) * Scale;


(* revision history
hm 22.2.2007		rev 1.2
	changed VAR RETAIN PERSISTENT to VAR RETAIN for better compatibility
	wago lon contollers do not support persisitent

*)
END_FUNCTION_BLOCK

(* POU click, ST *)
FUNCTION_BLOCK click
VAR_INPUT
	in : BOOL;
END_VAR
VAR_OUTPUT
	Q : BOOL;
	single : BOOL;
	double : BOOL;
	triple : BOOL;
	status: BYTE;
END_VAR
VAR_INPUT CONSTANT
	T_debounce : TIME := t#10ms;
	T_short : TIME := t#200ms;
	T_pause : TIME := t#500ms;
	T_reconfig : TIME := t#1m;
END_VAR
VAR
	debounce : TON;
	tx : TIME;
	last : TIME;
	init : BOOL;
	edge : BOOL;
	standby: BOOL;
	state: INT;
END_VAR

(*
version 1.2	15 sep 2007
programmer 	oscat
tested by		tobias

click checks an input for single, double or tripple click and sets the corresponding output single, doulbe or triple for the time the input stays high at the last click.
the maximum high and low time for a click can beconfigrured with setup variables.
the input cinfigures itself to be high or low active dependung on which state the input stays longer than t_reconfig.

*)
(* read system time *)
tx := DWORD_TO_TIME(T_PLC_MS());

(* set last and tx if never started before *)
IF NOT init THEN
	init := TRUE;
	last := tx;
	debounce.PT := T_debounce;
	standby := in;
END_IF;

(* debounce input *)
debounce(in := in XOR standby);
Q := debounce.Q;

(* delete outputs if input is inactive *)
IF NOT Q THEN
	single := FALSE;
	double := FALSE;
	triple := FALSE;
	status := 110;
END_IF;

(* check for input edge *)
IF Q XOR edge THEN
	edge := in;
	last := tx;
	IF Q THEN state := state + 1; END_IF;
END_IF;

IF (q AND tx - last >= T_short) OR (NOT q AND tx - last >= t_pause) THEN
	CASE state OF
		1:	single := TRUE;
			status := 111;
		2:	double := TRUE;
			status := 112;
		3:	triple := TRUE;
			status := 113;
	END_CASE;
	state := 0;
END_IF;

(* determine if high or low active *)
IF tx - last >= t_reconfig THEN
	standby := in;
	last := tx;
END_IF;



(* revision history

15 Feb 2007	rev 1.0	hm
	created original version

18.5.2007		rev 1.1 hm
	corrected an error while execution would stop after t_reconfig elapsed.

15.9.2007		rev 1.2 hm
	replaced Time() with T_PLC_MS for compatibility and performance reasons

*)
END_FUNCTION_BLOCK

(* POU CLK_1ms, ST *)
FUNCTION_BLOCK CLK_1ms
VAR_INPUT
END_VAR
VAR_OUTPUT
	Q : BOOL;
END_VAR
VAR
	CLK : BOOL;
	edge : BOOL := 0;
	stime: DWORD;
END_VAR

(*
version 1.1	17 sep 2007
programmer 	hugo
tested by		tobias

clk_gen uses the internal sps time to generate one pulse every 1 ms
every pulse is only valid for one cycle so that a edge trigger is not necessary
clk_gen generates pulses depending on the accuracy of the system clock.

be careful, 1ms clocks will only work on very powerful sps cpu's
wago 750 - 841 will work with pulse width >= 10ms
*)
stime := T_PLC_MS();
clk := stime.0;
Q := clk XOR edge;
edge := CLK;

(* revision history
hm	4. aug 2006		rev 1.0
	original version

hm	17. sep 2007	rev 1.1
	replaced time() with T_PLC_MS() for compatibility reasons

*)
END_FUNCTION_BLOCK

(* POU stime, ST *)
FUNCTION_BLOCK stime
VAR_INPUT
END_VAR
VAR_OUTPUT
	tx : DWORD;
END_VAR
VAR
	last_time: DWORD;
	bit31: BOOL;
END_VAR

(* this function block makes sure that the timer of a siemens sps counts from 0 - 2^32-1. *)
(* this FB is only necessary for siemens sps
the siemens sps timer counts from 0 to 2^31-1 and starts at 0 sfter overrun.
this means that the bit 31 (the highest bit ) will never be used and therefore
a problem arises when t2 - t1 is checked.
t2 - t1 is always valid also in an timer overrun situation where the time t1 is very high and t2 is very low.
the result of the subtraction t2 - t1 however is still valid.
this calculation does not work for soiemens because the highest bit is not used.

this module stores the highest bit, changes the highest bit at every overrun occurence and stuffs ther highest bit in the output.
the output is then used by t_plc_us and t_plc_ms.

the correction needs and fb and not a function because the value of the highest bit has to be stored.

do never use this function block in a codesys environment. the timer in codesys is correct and runs from 0 to 2^32-1
*)

(* read the system timer *)
tx := TIME_TO_DWORD(TIME());

(* check for overrun *)
IF tx < last_time THEN
	(* an overrun has occured, change the value of the highest bit *)
	bit31 := NOT bit31;
END_IF;

(* remember the last system time for the next overrun check *)
last_time := tx;

(* stuff the highest bit into the timer value *)
tx.31 := bit31;
END_FUNCTION_BLOCK

(* POU CLK_2ms, ST *)
FUNCTION_BLOCK CLK_2ms
VAR_INPUT
END_VAR
VAR_OUTPUT
	Q : BOOL;
END_VAR
VAR
	CLK : BOOL;
	edge : BOOL := 0;
	stime: DWORD;
END_VAR

(*
version 1.1	17 sep 2007
programmer 	hugo
tested by		tobias

clk_gen uses the internal sps time to generate one pulse every 2 ms
every pulse is only valid for one cycle so that a edge trigger is not necessary
clk_gen generates pulses depending on the accuracy of the system clock.

be careful, 1ms clocks will only work on very powerful sps cpu's
wago 750 - 841 will work with pulse width >= 10ms
*)
stime := T_PLC_MS();
clk := stime.1;
Q := clk XOR edge;
edge := CLK;

(* revision history
hm	4. aug 2006		rev 1.0
	original version

hm	17. sep 2007	rev 1.1
	replaced time() with T_PLC_MS() for compatibility reasons

*)
END_FUNCTION_BLOCK

(* POU CLK_4ms, ST *)
FUNCTION_BLOCK CLK_4ms
VAR_INPUT
END_VAR
VAR_OUTPUT
	Q : BOOL;
END_VAR
VAR
	CLK : BOOL;
	edge : BOOL := 0;
	stime: DWORD;
END_VAR

(*
version 1.1	17 sep 2007
programmer 	hugo
tested by		tobias

clk_gen uses the internal sps time to generate one pulse every 4 ms
every pulse is only valid for one cycle so that a edge trigger is not necessary
clk_gen generates pulses depending on the accuracy of the system clock.

be careful, 1ms clocks will only work on very powerful sps cpu's
wago 750 - 841 will work with pulse width >= 10ms
*)
stime := T_PLC_MS();
clk := stime.2;
Q := clk XOR edge;
edge := CLK;

(* revision history
hm	4. aug 2006		rev 1.0
	original version

hm	17. sep 2007	rev 1.1
	replaced time() with T_PLC_MS() for compatibility reasons

*)
END_FUNCTION_BLOCK

(* POU CLK_8ms, ST *)
FUNCTION_BLOCK CLK_8ms
VAR_INPUT
END_VAR
VAR_OUTPUT
	Q : BOOL;
END_VAR
VAR
	CLK : BOOL;
	edge : BOOL := 0;
	stime: DWORD;
END_VAR

(*
version 1.1	17 sep 2007
programmer 	hugo
tested by		tobias

clk_gen uses the internal sps time to generate one pulse every 8 ms
every pulse is only valid for one cycle so that a edge trigger is not necessary
clk_gen generates pulses depending on the accuracy of the system clock.

be careful, 1ms clocks will only work on very powerful sps cpu's
wago 750 - 841 will work with pulse width >= 10ms
*)
stime := T_PLC_MS();
clk := stime.3;
Q := clk XOR edge;
edge := CLK;

(* revision history
hm	4. aug 2006		rev 1.0
	original version

hm	17. sep 2007	rev 1.1
	replaced time() with T_PLC_MS() for compatibility reasons

*)
END_FUNCTION_BLOCK

(* POU clk_div, ST *)
FUNCTION_BLOCK clk_div
VAR_INPUT
	clk : BOOL;
	rst: BOOL;
END_VAR
VAR_OUTPUT
	Q0 : BOOL := 0;
	Q1 : BOOL := 0;
	Q2 : BOOL := 0;
	Q3 : BOOL := 0;
	Q4 : BOOL := 0;
	Q5 : BOOL := 0;
	Q6 : BOOL := 0;
	Q7 : BOOL := 0;
END_VAR
VAR
	cnt: BYTE := 0;
END_VAR

(*
version 1.0	4 aug 2006
programmer 	hugo
tested by		tobias

this is a clock divider
each output divides the signal by 2
Q0 = clk / 2 , Q1 = Q0 / 2 and so on.
the outputs have a 50% duty cycle each.


*)
IF clk AND NOT rst THEN
	cnt:= cnt +1;
	Q0 := cnt.0;
	Q1 := cnt.1;
	Q2 := cnt.2;
	Q3 := cnt.3;
	Q4 := cnt.4;
	Q5 := cnt.5;
	Q6 := cnt.6;
	Q7 := cnt.7;
END_IF;
IF rst THEN
	cnt:= 0;
	Q0 := 0;
	Q1 := 0;
	Q2 := 0;
	Q3 := 0;
	Q4 := 0;
	Q5 := 0;
	Q6 := 0;
	Q7 := 0;
END_IF;
END_FUNCTION_BLOCK

(* POU CLK_Prg, ST *)
	FUNCTION_BLOCK CLK_Prg
VAR_INPUT
	PT : TIME := t#10ms;
END_VAR
VAR_OUTPUT
	Q : BOOL := 0;
END_VAR
VAR
	init : BOOL := FALSE;
	last : TIME;
	tx: TIME;
END_VAR

(*
version 1.2	17 sep 2007
programmer 	hugo
tested by		tobias

clk_prg uses the internal sps time to generate a clock with programmable period time.
the period time is defined for 10ms .. 65s
the first cycle after start is a clk pulse and then depending on the programmed period time a delay.
every pulse is only valid for one cycle.
the accuracy of clk_prg is depending on the accuracy of the system clock.

*)
(* read system time *)
tx := DWORD_TO_TIME(T_PLC_MS());

(* initialize on startup *)
IF NOT init THEN
	init := TRUE;
	last := tx - pt;
END_IF;

(* generate output pulse when next_pulse is reached *)
IF tx - last >= pt THEN
	Q := TRUE;
	last := tx;
ELSE
	Q := FALSE;
END_IF;


(* revision hiostory

hm 25 feb 2007	rev 1.1
	rewritten code for higher performance
	pt can now be changed during runtime

hm	17. sep 2007	rev 1.2
	replaced time() with t_plc_ms() for compatibility reasons

*)
END_FUNCTION_BLOCK

(* POU CLK_Pulse, ST *)
FUNCTION_BLOCK CLK_Pulse
VAR_INPUT
	PT : TIME := t#10ms;
	N : INT := 0;
	rst : BOOL := 0;
END_VAR
VAR_OUTPUT
	Q : BOOL := 0;
	cnt : INT := 0;
	run : BOOL := 0;
END_VAR
VAR
	pti : TIME := t#0ms;
	next_pulse: TIME := T#0s;
	overflow: BOOL := FALSE;
	tx: TIME;
END_VAR

(*
version 1.1	17 sep 2007
programmer 	hugo
tested by		tobias

clk_pulse uses the internal sps time to generate a clock with programmable period time.
the period time is defined for 10ms .. 65s.
pulse generation is continuous if N = 0 and for n pulses otherwise.
if the period time is set to less then 10ms the min clock perid is 10ms.
the first cycle after start is a clk pulse and then depending on the programmed period time a delay.
every pulse is only valid for one cycle so that a edge trigger is not necessary
clk_prg depending on the accuracy of the system clock.

*)
(* read system *)
tx := DWORD_TO_TIME(T_PLC_MS());


IF rst THEN
	run := FALSE;
	pti := t#0ms;
	next_pulse := t#0ms;
	overflow := FALSE;
	Q := FALSE;
	cnt := 0;
ELSIF cnt <= N OR N = 0 THEN
	IF NOT run THEN
		next_pulse := tx;
		run := TRUE;
		IF pt < T#10ms THEN PTI := T#10ms; ELSE pti := pt; END_IF;
	END_IF;
	IF tx >= next_pulse AND NOT overflow AND (cnt < N OR N = 0) THEN
		Q := TRUE;
		cnt := cnt + 1;
		IF next_pulse + pti < next_pulse THEN
			overflow := TRUE;
		END_IF;
		next_pulse := next_pulse + pti;
	ELSE
		Q := FALSE;
		IF cnt = N THEN run := FALSE; END_IF
		IF tx <= next_pulse THEN overflow := FALSE; END_IF;
	END_IF;
END_IF

(* revision history
hm		4. aug 2006		rev 1.0
	original version

hm		17. sep 2007	rev 1.1
	replaced time() with T_PLC_S() fr compatblity reasons

*)
END_FUNCTION_BLOCK

(* POU compatibility, ST *)
FUNCTION_BLOCK compatibility
VAR_INPUT
END_VAR
VAR_OUTPUT
END_VAR
VAR
END_VAR

(*
	version 1.0	16 sep 2007
	programmer 	oscat
	tested BY		oscat

METER measures usage of power or similar values the output MX is the summ of the inputs over time.
MX := sum over time of I1 * P1 + I2 * P2.
a simple example is the consumption counter for a 2 stage oil burner where stage 1 is 10KW and stage 2 is 20KW.
I1 and I2 decide which value is accounted for, I1 = True only counts P1, I2 is True counts P2 
and I1 and I2 is true counts P1 and P2.
the meter can be used for all kind of consumption meters. P1 and P2 can change on the fly.

*)
RETURN;
END_FUNCTION_BLOCK

(* POU D_Trig, ST *)
FUNCTION_BLOCK D_Trig
VAR_INPUT
	in : DWORD;
END_VAR
VAR_OUTPUT
	Q : BOOL;
	X : DWORD;
END_VAR
VAR
	last_in : DWORD;
END_VAR

(*
version 1.0	4 Sep 2007
programmer 	hugo
tested by		tobias

this block is similar to the IEC Standard R_trig and F_trig but it monitors a DWORD, WORD or Byte Variable instead and generated an Output Pulse for one cycle only when the input has changed.
an additional output x (Dword) will state the chage of the input.
Example: the input has chaged from 0001 to 0010 then the output x will be 2.

*)
IF (in XOR last_in) <> 0 THEN
	Q := TRUE;
	X := in - last_in;
	last_in := in;
ELSE
	Q := FALSE;
END_IF;


(* revision history

hm 4.09.2007	rev 1.0
	original version released

*)
END_FUNCTION_BLOCK

(* POU date_test, ST *)
FUNCTION_BLOCK date_test
VAR_INPUT
END_VAR
VAR_OUTPUT
END_VAR
VAR
	dout: DT;
	x: DWORD;
	y: INT;
	dez: BOOL := TRUE;
	d: INT;
	l : BOOL;
END_VAR
dout := DWORD_TO_DT(x);
y := year(DWORD_TO_DATE(x));
d := day_of_month(DWORD_TO_DATE(x));
l := leap_of_Date(DWORD_TO_DATE(x));


(* prepare next date *)

IF dez THEN
	x := DATE_TO_DWORD(date_add(DWORD_TO_DATE(x),0,0,1,1))-1;
	dez := FALSE;
ELSE
	x := x + 1;
	dez := TRUE;
END_IF;
END_FUNCTION_BLOCK

(* POU day_to_time, ST *)
FUNCTION day_to_time : TIME
VAR_INPUT
	input : REAL;
END_VAR
VAR
END_VAR

(*
version 1.0	4 aug 2006
programmer 	hugo
tested by		tobias

converts an amount of days in real to time 
*)
day_to_time := DWORD_TO_TIME(REAL_TO_DWORD(input * 86400000));
END_FUNCTION

(* POU DCF77, ST *)
FUNCTION_BLOCK DCF77
VAR_INPUT
	rec : BOOL;
END_VAR
VAR_INPUT CONSTANT
	sync_timeout : TIME := t#2m;
	time_offset : TIME := t#1h;
	dst_en : BOOL := TRUE;
END_VAR
VAR_OUTPUT
	TP : BOOL;
	DST : BOOL;
	weekday : INT;
	error: BOOL := TRUE;
	RTC : DT;
	RTC1 : DT;
	msec : INT;
	sync : BOOL;
END_VAR
VAR
	MEZ : DT;
	UTC : DT;
	state : INT;
	edge: BOOL;
	tx : TIME;
	ty: TIME;
	last : TIME;
	bits : ARRAY[0..58] OF BOOL;
	cnt : INT;
	i : INT;
	old_time : DT;
	minute : INT;
	hour : INT;
	day : INT;
	month : INT;
	year : INT;
	last_sync: TIME;
	t1: TIME;
END_VAR


(*
version 1.3	17 sep 2007
programmer 	hugo
tested by		tobias

